C03637=1085.403,192.543,-73.156,175.423,21.883,153.539
C03638=1085.409,192.792,-73.179,175.426,21.885,153.539
C03639=1085.415,193.041,-73.202,175.428,21.886,153.539
C03640=1085.420,193.290,-73.225,175.431,21.888,153.539
C03641=1085.425,193.539,-73.248,175.433,21.890,153.539
C03642=1085.431,193.787,-73.272,175.436,21.892,153.539
C03643=1085.437,194.036,-73.295,175.438,21.893,153.539
C03644=1085.443,194.285,-73.318,175.441,21.895,153.539
C03645=1085.448,194.534,-73.342,175.443,21.897,153.539
C03646=1085.453,194.783,-73.364,175.446,21.899,153.539
C03647=1085.459,195.032,-73.387,175.448,21.900,153.539
C03648=1085.465,195.280,-73.411,175.451,21.902,153.539
C03649=1085.470,195.530,-73.435,175.453,21.904,153.539
C03650=1085.476,195.779,-73.458,175.457,21.906,153.539
C03651=1085.482,196.027,-73.481,175.459,21.907,153.539
C03652=1085.487,196.277,-73.504,175.461,21.909,153.539
C03653=1085.493,196.525,-73.528,175.464,21.911,153.539
C03654=1085.498,196.774,-73.551,175.467,21.912,153.539
C03655=1085.504,197.023,-73.574,175.469,21.914,153.539
C03656=1085.510,197.271,-73.598,175.471,21.916,153.539
C03657=1085.515,197.520,-73.621,175.474,21.917,153.539
C03658=1085.521,197.769,-73.644,175.476,21.919,153.539
C03659=1085.526,198.018,-73.667,175.479,21.921,153.539
C03660=1085.532,198.267,-73.691,175.482,21.923,153.539
C03661=1085.538,198.515,-73.714,175.485,21.925,153.539
C03662=1085.543,198.765,-73.737,175.487,21.927,153.539
C03663=1085.549,199.013,-73.761,175.490,21.928,153.539
C03664=1085.554,199.262,-73.784,175.492,21.930,153.539
C03665=1085.560,199.510,-73.808,175.495,21.932,153.539
C03666=1085.566,199.759,-73.831,175.497,21.933,153.539
C03667=1085.572,200.009,-73.855,175.500,21.935,153.539
C03668=1085.577,200.258,-73.879,175.502,21.937,153.539
C03669=1085.583,200.506,-73.902,175.505,21.938,153.539
C03670=1085.589,200.755,-73.925,175.508,21.940,153.539
C03671=1085.594,201.004,-73.949,175.511,21.942,153.538
C03672=1085.600,201.252,-73.973,175.513,21.944,153.539
C03673=1085.605,201.501,-73.996,175.516,21.945,153.539
C03674=1085.612,201.750,-74.020,175.518,21.947,153.538
C03675=1085.617,201.999,-74.043,175.521,21.949,153.538
C03676=1085.623,202.248,-74.067,175.523,21.950,153.538
C03677=1085.628,202.497,-74.090,175.526,21.952,153.538
C03678=1085.634,202.745,-74.115,175.529,21.954,153.538
C03679=1085.639,202.994,-74.138,175.532,21.956,153.538
C03680=1085.645,203.243,-74.162,175.534,21.957,153.538
C03681=1085.651,203.492,-74.185,175.537,21.959,153.538
C03682=1085.656,203.741,-74.209,175.539,21.961,153.538
C03683=1085.661,203.990,-74.233,175.542,21.963,153.538
C03684=1085.667,204.239,-74.257,175.544,21.964,153.538
C03685=1085.673,204.487,-74.281,175.548,21.966,153.538
C03686=1085.678,204.736,-74.304,175.550,21.968,153.538
C03687=1085.684,204.985,-74.328,175.553,21.970,153.538
C03688=1085.689,205.233,-74.352,175.555,21.972,153.538
C03689=1085.695,205.483,-74.376,175.558,21.973,153.538
C03690=1085.701,205.731,-74.400,175.560,21.975,153.538
C03691=1085.706,205.980,-74.424,175.564,21.977,153.538
C03692=1085.712,206.229,-74.447,175.566,21.979,153.538
C03693=1085.717,206.477,-74.471,175.568,21.981,153.538
C03694=1085.724,206.726,-74.495,175.571,21.983,153.538
C03695=1085.729,206.976,-74.519,175.574,21.984,153.538
C03696=1085.734,207.224,-74.543,175.576,21.986,153.538
C03697=1085.757,208.251,-74.642,175.658,22.028,153.535
C03698=1085.767,208.639,-74.680,175.662,22.033,153.535
C03699=1085.775,209.027,-74.718,175.666,22.037,153.535
C03700=1085.783,209.415,-74.756,175.670,22.041,153.536
C03701=1085.793,209.803,-74.795,175.673,22.045,153.536
C03702=1085.798,210.051,-74.819,175.676,22.048,153.536
C03703=1085.804,210.301,-74.843,175.678,22.050,153.536
C03704=1085.810,210.549,-74.868,175.681,22.053,153.536
C03705=1085.815,210.798,-74.892,175.684,22.056,153.537
C03706=1085.821,211.047,-74.917,175.686,22.058,153.537
C03707=1085.826,211.295,-74.942,175.689,22.061,153.537
C03708=1085.832,211.544,-74.966,175.691,22.064,153.537
C03709=1085.838,211.793,-74.990,175.694,22.067,153.538
C03710=1085.843,212.042,-75.015,175.696,22.069,153.538
C03711=1085.849,212.290,-75.040,175.699,22.072,153.538
C03712=1085.854,212.539,-75.064,175.701,22.075,153.538
C03713=1085.860,212.788,-75.089,175.704,22.077,153.538
C03714=1085.866,213.036,-75.114,175.707,22.080,153.538
C03715=1085.872,213.285,-75.138,175.709,22.083,153.539
C03716=1085.877,213.534,-75.163,175.712,22.086,153.539
C03717=1085.882,213.784,-75.188,175.714,22.088,153.539
C03718=1085.888,214.032,-75.213,175.716,22.091,153.539
C03719=1085.894,214.281,-75.238,175.720,22.094,153.539
C03720=1085.899,214.529,-75.263,175.722,22.096,153.540
C03721=1085.905,214.777,-75.287,175.725,22.099,153.540
C03722=1085.910,215.027,-75.311,175.727,22.102,153.540
C03723=1085.916,215.275,-75.336,175.730,22.105,153.540
C03724=1085.921,215.524,-75.362,175.732,22.107,153.540
C03725=1085.927,215.772,-75.387,175.734,22.110,153.541
C03726=1085.933,216.022,-75.411,175.737,22.113,153.541
C03727=1085.938,216.270,-75.436,175.740,22.115,153.541
C03728=1085.944,216.519,-75.461,175.743,22.118,153.541
C03729=1085.949,216.767,-75.486,175.745,22.121,153.541
C03730=1085.955,217.016,-75.511,175.748,22.124,153.542
C03731=1085.961,217.264,-75.536,175.750,22.126,153.542
C03732=1085.967,217.514,-75.561,175.753,22.129,153.542
C03733=1085.973,217.762,-75.586,175.755,22.132,153.542
C03734=1085.977,218.011,-75.611,175.757,22.134,153.542
C03735=1085.984,218.260,-75.636,175.761,22.137,153.543
C03736=1085.989,218.508,-75.660,175.763,22.139,153.543
C03737=1085.995,218.757,-75.686,175.766,22.143,153.543
C03738=1086.000,219.006,-75.710,175.768,22.145,153.543
C03739=1086.006,219.255,-75.736,175.771,22.148,153.543
C03740=1086.012,219.503,-75.761,175.773,22.151,153.544
C03741=1086.017,219.752,-75.785,175.776,22.153,153.544
C03742=1086.023,220.001,-75.811,175.779,22.156,153.544
C03743=1086.028,220.249,-75.836,175.782,22.159,153.544
C03744=1086.034,220.498,-75.861,175.784,22.161,153.544
C03745=1086.040,220.747,-75.886,175.786,22.164,153.544
C03746=1086.046,220.995,-75.911,175.789,22.167,153.545
C03747=1086.051,221.244,-75.937,175.791,22.169,153.545
C03748=1086.057,221.493,-75.962,175.794,22.172,153.545
C03749=1086.063,221.741,-75.987,175.797,22.175,153.545
C03750=1086.072,222.133,-76.027,175.801,22.179,153.546
C03751=1086.081,222.526,-76.066,175.805,22.183,153.546
C03752=1086.090,222.917,-76.107,175.809,22.188,153.546
C03753=1086.098,223.309,-76.146,175.813,22.192,153.547
C03754=1086.103,223.558,-76.172,175.816,22.195,153.547
C03755=1086.109,223.806,-76.197,175.818,22.197,153.547
C03756=1086.115,224.054,-76.222,175.821,22.201,153.547
C03757=1086.121,224.303,-76.248,175.824,22.203,153.547
C03758=1086.126,224.553,-76.273,175.827,22.206,153.548
C03759=1086.131,224.801,-76.298,175.829,22.209,153.548
C03760=1086.138,225.050,-76.324,175.832,22.211,153.548
C03761=1086.143,225.298,-76.350,175.834,22.214,153.548
C03762=1086.149,225.546,-76.375,175.837,22.217,153.548
C03763=1086.154,225.795,-76.401,175.839,22.219,153.548
C03764=1086.160,226.044,-76.426,175.842,22.223,153.549
C03765=1086.165,226.292,-76.452,175.845,22.225,153.549
C03766=1086.171,226.541,-76.477,175.848,22.228,153.549
C03767=1086.177,226.790,-76.503,175.850,22.231,153.549
C03768=1086.182,227.039,-76.529,175.853,22.233,153.549
C03769=1086.188,227.287,-76.554,175.855,22.236,153.550
C03770=1086.193,227.536,-76.580,175.858,22.239,153.550
C03771=1086.200,227.785,-76.605,175.860,22.241,153.550
C03772=1086.205,228.034,-76.631,175.863,22.245,153.550
C03773=1086.211,228.282,-76.656,175.866,22.247,153.551
C03774=1086.216,228.531,-76.682,175.869,22.250,153.551
C03775=1086.222,228.779,-76.707,175.871,22.252,153.551
C03776=1086.228,229.028,-76.733,175.874,22.255,153.551
C03777=1086.234,229.277,-76.760,175.876,22.258,153.551
C03778=1086.239,229.525,-76.785,175.879,22.261,153.552
C03779=1086.245,229.774,-76.811,175.881,22.263,153.552
C03780=1086.251,230.022,-76.836,175.885,22.266,153.552
C03781=1086.256,230.271,-76.862,175.887,22.269,153.552
C03782=1086.262,230.520,-76.888,175.890,22.272,153.552
C03783=1086.267,230.768,-76.913,175.892,22.274,153.552
C03784=1086.273,231.016,-76.939,175.895,22.277,153.553
C03785=1086.279,231.265,-76.965,175.898,22.280,153.553
C03786=1086.284,231.514,-76.991,175.900,22.283,153.553
C03787=1086.290,231.763,-77.017,175.903,22.285,153.553
C03788=1086.295,232.011,-77.043,175.905,22.288,153.554
C03789=1086.301,232.260,-77.069,175.909,22.291,153.554
C03790=1086.306,232.509,-77.095,175.911,22.293,153.554
C03791=1086.313,232.757,-77.120,175.914,22.297,153.554
C03792=1086.318,233.006,-77.147,175.916,22.299,153.554
C03793=1086.324,233.255,-77.173,175.919,22.302,153.555
C03794=1086.329,233.503,-77.198,175.921,22.305,153.555
C03795=1086.335,233.751,-77.224,175.924,22.307,153.555
C03796=1086.341,234.000,-77.250,175.927,22.310,153.555
C03797=1086.346,234.248,-77.277,175.930,22.313,153.555
C03798=1086.352,234.497,-77.303,175.933,22.316,153.556
C03799=1086.357,234.746,-77.329,175.935,22.319,153.556
C03800=1086.363,234.995,-77.355,175.938,22.322,153.556
C03801=1086.368,235.243,-77.381,175.940,22.324,153.556
C03802=1086.377,235.626,-77.421,175.945,22.329,153.556
C03803=1086.386,236.010,-77.462,175.948,22.333,153.557
C03804=1086.394,236.393,-77.502,175.953,22.337,153.557
C03805=1086.404,236.777,-77.542,175.957,22.341,153.557
C03806=1086.409,237.025,-77.569,175.960,22.344,153.558
C03807=1086.414,237.273,-77.595,175.962,22.347,153.558
C03808=1086.420,237.522,-77.621,175.965,22.350,153.558
C03809=1086.425,237.771,-77.647,175.968,22.353,153.558
C03810=1086.431,238.019,-77.674,175.970,22.355,153.558
C03811=1086.437,238.267,-77.700,175.973,22.359,153.559
C03812=1086.442,238.516,-77.726,175.976,22.361,153.559
C03813=1086.448,238.765,-77.753,175.979,22.364,153.559
C03814=1086.454,239.014,-77.779,175.981,22.366,153.559
C03815=1086.459,239.262,-77.806,175.984,22.369,153.559
C03816=1086.465,239.510,-77.832,175.987,22.372,153.560
C03817=1086.471,239.759,-77.858,175.989,22.375,153.560
C03818=1086.476,240.008,-77.885,175.992,22.378,153.560
C03819=1086.482,240.256,-77.912,175.994,22.380,153.560
C03820=1086.488,240.505,-77.937,175.998,22.383,153.560
C03821=1086.493,240.753,-77.964,176.001,22.386,153.561
C03822=1086.499,241.002,-77.991,176.003,22.389,153.561
C03823=1086.505,241.250,-78.017,176.006,22.391,153.561
C03824=1086.510,241.499,-78.043,176.008,22.394,153.561
C03825=1086.516,241.747,-78.070,176.011,22.397,153.561
C03826=1086.522,241.996,-78.097,176.014,22.400,153.562
C03827=1086.528,242.244,-78.123,176.016,22.403,153.562
C03828=1086.533,242.493,-78.149,176.019,22.406,153.562
C03829=1086.539,242.742,-78.176,176.022,22.408,153.562
C03830=1086.545,242.990,-78.202,176.025,22.411,153.563
C03831=1086.551,243.238,-78.229,176.028,22.414,153.563
C03832=1086.556,243.488,-78.257,176.030,22.417,153.563
C03833=1086.562,243.736,-78.283,176.033,22.420,153.563
C03834=1086.568,243.984,-78.310,176.035,22.422,153.563
C03835=1086.573,244.233,-78.336,176.038,22.425,153.564
C03836=1086.579,244.482,-78.363,176.041,22.428,153.564
C03837=1086.584,244.730,-78.390,176.043,22.431,153.564
C03838=1086.590,244.979,-78.417,176.047,22.434,153.564
C03839=1086.596,245.227,-78.443,176.050,22.437,153.565
C03840=1086.601,245.475,-78.470,176.052,22.439,153.565
C03841=1086.606,245.724,-78.497,176.055,22.443,153.565
C03842=1086.612,245.972,-78.524,176.057,22.445,153.565
C03843=1086.618,246.221,-78.550,176.060,22.448,153.565
C03844=1086.623,246.470,-78.578,176.063,22.451,153.566
C03845=1086.629,246.718,-78.604,176.065,22.454,153.566
C03846=1086.635,246.967,-78.631,176.069,22.456,153.566
C03847=1086.641,247.215,-78.658,176.071,22.460,153.566
C03848=1086.646,247.464,-78.685,176.074,22.462,153.566
C03849=1086.652,247.712,-78.712,176.077,22.465,153.567
C03850=1086.657,247.961,-78.739,176.080,22.468,153.567
C03851=1086.663,248.209,-78.766,176.082,22.471,153.567
C03852=1086.668,248.457,-78.794,176.085,22.474,153.567
C03853=1086.674,248.706,-78.820,176.087,22.476,153.568
C03854=1086.682,249.083,-78.861,176.092,22.481,153.568
C03855=1086.690,249.459,-78.902,176.096,22.486,153.568
C03856=1086.699,249.835,-78.943,176.100,22.490,153.569
C03857=1086.707,250.211,-78.984,176.105,22.494,153.569
C03858=1086.712,250.460,-79.012,176.107,22.497,153.569
C03859=1086.719,250.709,-79.039,176.110,22.500,153.569
C03860=1086.724,250.957,-79.067,176.113,22.503,153.570
C03861=1086.730,251.206,-79.093,176.115,22.506,153.570
C03862=1086.735,251.454,-79.120,176.118,22.509,153.570
C03863=1086.741,251.703,-79.147,176.121,22.512,153.570
C03864=1086.746,251.951,-79.175,176.123,22.514,153.571
C03865=1086.752,252.200,-79.202,176.126,22.518,153.571
C03866=1086.758,252.448,-79.229,176.129,22.520,153.571
C03867=1086.764,252.696,-79.257,176.132,22.523,153.571
C03868=1086.769,252.945,-79.284,176.135,22.526,153.571
C03869=1086.774,253.193,-79.311,176.138,22.529,153.572
C03870=1086.780,253.442,-79.339,176.140,22.532,153.572
C03871=1086.785,253.691,-79.366,176.143,22.535,153.572
C03872=1086.791,253.938,-79.393,176.146,22.538,153.572
C03873=1086.796,254.187,-79.421,176.148,22.540,153.573
C03874=1086.803,254.435,-79.448,176.151,22.543,153.573
C03875=1086.808,254.684,-79.476,176.154,22.546,153.573
C03876=1086.814,254.932,-79.504,176.156,22.549,153.573
C03877=1086.820,255.181,-79.531,176.160,22.552,153.574
C03878=1086.825,255.430,-79.558,176.163,22.555,153.574
C03879=1086.831,255.678,-79.585,176.165,22.558,153.574
C03880=1086.836,255.926,-79.613,176.168,22.561,153.574
C03881=1086.842,256.175,-79.641,176.171,22.564,153.575
C03882=1086.848,256.423,-79.668,176.174,22.567,153.575
C03883=1086.853,256.671,-79.695,176.176,22.569,153.575
C03884=1086.860,256.920,-79.723,176.179,22.572,153.575
C03885=1086.865,257.169,-79.750,176.182,22.575,153.575
C03886=1086.870,257.417,-79.778,176.184,22.578,153.576
C03887=1086.877,257.665,-79.806,176.187,22.581,153.576
C03888=1086.882,257.914,-79.833,176.190,22.584,153.576
C03889=1086.887,258.162,-79.861,176.193,22.586,153.576
C03890=1086.894,258.410,-79.889,176.196,22.590,153.577
C03891=1086.899,258.659,-79.916,176.199,22.592,153.577
C03892=1086.905,258.908,-79.945,176.202,22.596,153.577
C03893=1086.911,259.155,-79.972,176.204,22.598,153.577
C03894=1086.916,259.404,-79.999,176.207,22.601,153.577
C03895=1086.922,259.653,-80.028,176.210,22.604,153.578
C03896=1086.928,259.900,-80.055,176.212,22.607,153.578
C03897=1086.934,260.149,-80.083,176.216,22.609,153.578
C03898=1086.939,260.398,-80.110,176.219,22.613,153.578
C03899=1086.945,260.646,-80.138,176.222,22.616,153.579
C03900=1086.951,260.894,-80.166,176.224,22.618,153.579
C03901=1086.956,261.142,-80.194,176.227,22.621,153.579
C03902=1086.963,261.391,-80.222,176.230,22.624,153.579
C03903=1086.968,261.640,-80.249,176.233,22.627,153.579
C03904=1086.974,261.888,-80.277,176.235,22.630,153.580
C03905=1086.979,262.136,-80.305,176.238,22.633,153.580
C03906=1086.989,262.510,-80.347,176.243,22.638,153.580
C03907=1086.997,262.883,-80.390,176.247,22.641,153.581
C03908=1087.006,263.257,-80.431,176.251,22.646,153.581
C03909=1087.014,263.630,-80.474,176.256,22.650,153.581
C03910=1087.021,263.879,-80.501,176.258,22.653,153.581
C03911=1087.026,264.127,-80.529,176.261,22.656,153.582
C03912=1087.032,264.376,-80.557,176.264,22.659,153.582
C03913=1087.037,264.624,-80.585,176.266,22.662,153.582
C03914=1087.043,264.873,-80.613,176.269,22.665,153.582
C03915=1087.049,265.120,-80.642,176.272,22.668,153.583
C03916=1087.055,265.369,-80.670,176.276,22.671,153.583
C03917=1087.060,265.617,-80.698,176.279,22.674,153.583
C03918=1087.066,265.866,-80.727,176.281,22.677,153.583
C03919=1087.072,266.114,-80.755,176.284,22.680,153.584
C03920=1087.078,266.363,-80.783,176.287,22.683,153.584
C03921=1087.083,266.611,-80.811,176.290,22.686,153.584
C03922=1087.089,266.859,-80.839,176.292,22.689,153.584
C03923=1087.094,267.107,-80.867,176.295,22.691,153.585
C03924=1087.100,267.356,-80.896,176.298,22.695,153.585
C03925=1087.106,267.604,-80.924,176.301,22.698,153.585
C03926=1087.112,267.852,-80.953,176.303,22.700,153.585
C03927=1087.117,268.100,-80.981,176.306,22.703,153.586
C03928=1087.123,268.349,-81.009,176.309,22.707,153.586
C03929=1087.129,268.598,-81.037,176.312,22.710,153.586
C03930=1087.135,268.845,-81.066,176.315,22.713,153.586
C03931=1087.141,269.094,-81.094,176.318,22.715,153.587
C03932=1087.145,269.343,-81.123,176.321,22.719,153.587
C03933=1087.151,269.591,-81.152,176.324,22.721,153.587
C03934=1087.157,269.839,-81.180,176.327,22.725,153.587
C03935=1087.163,270.087,-81.208,176.329,22.727,153.588
C03936=1087.169,270.336,-81.236,176.332,22.731,153.588
C03937=1087.174,270.584,-81.265,176.335,22.733,153.588
C03938=1087.180,270.832,-81.293,176.338,22.737,153.588
C03939=1087.185,271.080,-81.323,176.341,22.740,153.589
C03940=1087.191,271.329,-81.351,176.343,22.743,153.589
C03941=1087.197,271.578,-81.379,176.346,22.745,153.589
C03942=1087.203,271.825,-81.408,176.349,22.749,153.589
C03943=1087.209,272.074,-81.436,176.352,22.752,153.590
C03944=1087.214,272.322,-81.466,176.355,22.755,153.590
C03945=1087.219,272.570,-81.494,176.357,22.758,153.590
C03946=1087.226,272.818,-81.523,176.361,22.760,153.590
C03947=1087.231,273.066,-81.551,176.364,22.764,153.591
C03948=1087.237,273.315,-81.581,176.367,22.767,153.591
C03949=1087.242,273.564,-81.609,176.370,22.770,153.591
C03950=1087.248,273.811,-81.638,176.372,22.772,153.591
C03951=1087.254,274.060,-81.666,176.375,22.776,153.592
C03952=1087.260,274.308,-81.696,176.378,22.779,153.592
C03953=1087.265,274.556,-81.723,176.381,22.782,153.592
C03954=1087.270,274.805,-81.753,176.384,22.785,153.593
C03955=1087.276,275.054,-81.781,176.387,22.789,153.593
C03956=1087.282,275.301,-81.810,176.389,22.791,153.593
C03957=1087.288,275.549,-81.840,176.392,22.794,153.593
C03958=1087.296,275.926,-81.883,176.397,22.799,153.594
C03959=1087.304,276.302,-81.927,176.401,22.804,153.594
C03960=1087.313,276.678,-81.970,176.406,22.808,153.594
C03961=1087.322,277.055,-82.015,176.409,22.813,153.595
C03962=1087.328,277.303,-82.044,176.412,22.816,153.595
C03963=1087.333,277.552,-82.073,176.415,22.819,153.596
C03964=1087.339,277.800,-82.102,176.419,22.822,153.596
C03965=1087.345,278.049,-82.131,176.422,22.825,153.596
C03966=1087.351,278.296,-82.160,176.425,22.828,153.596
C03967=1087.356,278.544,-82.190,176.427,22.831,153.597
C03968=1087.362,278.793,-82.218,176.430,22.834,153.597
C03969=1087.368,279.042,-82.247,176.433,22.838,153.597
C03970=1087.373,279.289,-82.276,176.436,22.841,153.597
C03971=1087.379,279.537,-82.306,176.439,22.844,153.598
C03972=1087.385,279.786,-82.335,176.442,22.847,153.598
C03973=1087.390,280.034,-82.364,176.445,22.851,153.598
C03974=1087.396,280.281,-82.393,176.447,22.853,153.598
C03975=1087.402,280.530,-82.423,176.450,22.856,153.599
C03976=1087.408,280.779,-82.451,176.453,22.859,153.599
C03977=1087.413,281.027,-82.481,176.456,22.862,153.599
C03978=1087.419,281.275,-82.510,176.459,22.866,153.600
C03979=1087.424,281.523,-82.539,176.462,22.869,153.600
C03980=1087.431,281.771,-82.568,176.465,22.872,153.600
C03981=1087.436,282.020,-82.598,176.467,22.875,153.601
C03982=1087.442,282.268,-82.627,176.470,22.878,153.601
C03983=1087.448,282.516,-82.656,176.473,22.881,153.601
C03984=1087.453,282.764,-82.686,176.476,22.884,153.601
C03985=1087.458,283.012,-82.715,176.479,22.888,153.602
C03986=1087.464,283.260,-82.746,176.482,22.891,153.602
C03987=1087.470,283.508,-82.775,176.485,22.894,153.602
C03988=1087.476,283.757,-82.804,176.488,22.897,153.603
C03989=1087.481,284.005,-82.834,176.491,22.900,153.603
C03990=1087.487,284.253,-82.863,176.493,22.903,153.603
C03991=1087.492,284.501,-82.892,176.496,22.907,153.604
C03992=1087.498,284.749,-82.922,176.499,22.910,153.604
C03993=1087.503,284.998,-82.952,176.502,22.913,153.604
C03994=1087.510,285.245,-82.981,176.505,22.917,153.604
C03995=1087.516,285.494,-83.011,176.508,22.920,153.605
C03996=1087.521,285.742,-83.041,176.511,22.923,153.605
C03997=1087.527,285.990,-83.070,176.514,22.926,153.605
C03998=1087.533,286.238,-83.100,176.517,22.929,153.606
C03999=1087.538,286.486,-83.129,176.519,22.932,153.606
C04000=1087.544,286.734,-83.159,176.522,22.935,153.606
C04001=1087.549,286.983,-83.188,176.525,22.939,153.606
C04002=1087.556,287.230,-83.218,176.528,22.942,153.607
C04003=1087.561,287.479,-83.248,176.531,22.945,153.607
C04004=1087.567,287.727,-83.278,176.534,22.948,153.607
C04005=1087.572,287.975,-83.308,176.537,22.951,153.608
C04006=1087.579,288.223,-83.337,176.540,22.955,153.608
C04007=1087.584,288.472,-83.367,176.544,22.958,153.608
C04008=1087.590,288.719,-83.397,176.547,22.961,153.608
C04009=1087.596,288.968,-83.427,176.549,22.965,153.609
C04010=1087.604,289.354,-83.473,176.554,22.969,153.609
C04011=1087.613,289.740,-83.520,176.558,22.974,153.610
C04012=1087.622,290.125,-83.566,176.563,22.979,153.610
C04013=1087.631,290.511,-83.613,176.567,22.984,153.611
C04014=1087.636,290.760,-83.643,176.570,22.988,153.611
C04015=1087.642,291.007,-83.673,176.573,22.991,153.611
C04016=1087.648,291.256,-83.703,176.576,22.994,153.612
C04017=1087.654,291.504,-83.733,176.579,22.998,153.612
C04018=1087.660,291.752,-83.762,176.582,23.001,153.612
C04019=1087.666,292.000,-83.792,176.585,23.004,153.613
C04020=1087.671,292.248,-83.822,176.588,23.007,153.613
C04021=1087.677,292.496,-83.852,176.591,23.011,153.613
C04022=1087.682,292.744,-83.883,176.594,23.014,153.614
C04023=1087.688,292.992,-83.913,176.597,23.017,153.614
C04024=1087.694,293.241,-83.944,176.599,23.020,153.614
C04025=1087.700,293.489,-83.974,176.602,23.024,153.615
C04026=1087.705,293.737,-84.004,176.605,23.027,153.615
C04027=1087.711,293.985,-84.034,176.608,23.030,153.615
C04028=1087.717,294.233,-84.064,176.611,23.033,153.615
C04029=1087.723,294.481,-84.095,176.614,23.037,153.616
C04030=1087.728,294.729,-84.124,176.617,23.040,153.616
C04031=1087.734,294.977,-84.155,176.620,23.043,153.616
C04032=1087.740,295.225,-84.185,176.623,23.046,153.617
C04033=1087.746,295.473,-84.215,176.626,23.050,153.617
C04034=1087.751,295.721,-84.245,176.629,23.053,153.617
C04035=1087.757,295.969,-84.275,176.632,23.057,153.618
C04036=1087.763,296.218,-84.307,176.635,23.060,153.618
C04037=1087.769,296.466,-84.337,176.638,23.063,153.618
C04038=1087.774,296.713,-84.367,176.641,23.067,153.619
C04039=1087.780,296.961,-84.398,176.644,23.070,153.619
C04040=1087.786,297.209,-84.428,176.647,23.073,153.619
C04041=1087.791,297.458,-84.458,176.650,23.077,153.620
C04042=1087.797,297.706,-84.489,176.653,23.080,153.620
C04043=1087.803,297.954,-84.519,176.656,23.084,153.620
C04044=1087.809,298.202,-84.550,176.659,23.087,153.621
C04045=1087.814,298.450,-84.581,176.662,23.090,153.621
C04046=1087.820,298.698,-84.611,176.665,23.094,153.621
C04047=1087.825,298.946,-84.642,176.667,23.097,153.622
C04048=1087.831,299.194,-84.672,176.670,23.101,153.622
C04049=1087.837,299.442,-84.703,176.673,23.104,153.623
C04050=1087.842,299.690,-84.734,176.676,23.108,153.623
C04051=1087.847,299.938,-84.764,176.679,23.111,153.623
C04052=1087.853,300.186,-84.796,176.682,23.115,153.624
C04053=1087.859,300.434,-84.826,176.685,23.118,153.624
C04054=1087.864,300.682,-84.857,176.688,23.121,153.624
C04055=1087.870,300.930,-84.888,176.691,23.125,153.625
C04056=1087.876,301.177,-84.918,176.694,23.128,153.625
C04057=1087.881,301.426,-84.949,176.697,23.132,153.626
C04058=1087.887,301.674,-84.980,176.700,23.135,153.626
C04059=1087.893,301.922,-85.011,176.703,23.139,153.626
C04060=1087.899,302.169,-85.042,176.706,23.142,153.627
C04061=1087.904,302.418,-85.073,176.708,23.146,153.627
C04062=1087.913,302.818,-85.122,176.714,23.152,153.628
C04063=1087.922,303.217,-85.172,176.718,23.157,153.628
C04064=1087.932,303.618,-85.222,176.723,23.163,153.629
C04065=1087.940,304.018,-85.272,176.728,23.168,153.629
C04066=1087.946,304.265,-85.303,176.731,23.172,153.630
C04067=1087.952,304.514,-85.335,176.734,23.175,153.630
C04068=1087.958,304.762,-85.365,176.737,23.179,153.631
C04069=1087.963,305.010,-85.396,176.740,23.183,153.631
C04070=1087.969,305.257,-85.427,176.743,23.186,153.631
C04071=1087.975,305.506,-85.458,176.746,23.189,153.632
C04072=1087.981,305.753,-85.489,176.749,23.193,153.632
C04073=1087.986,306.001,-85.520,176.752,23.196,153.632
C04074=1087.992,306.250,-85.552,176.755,23.200,153.633
C04075=1087.998,306.497,-85.583,176.758,23.203,153.633
C04076=1088.003,306.745,-85.614,176.761,23.207,153.634
C04077=1088.010,306.993,-85.645,176.764,23.210,153.634
C04078=1088.015,307.241,-85.676,176.767,23.214,153.634
C04079=1088.021,307.488,-85.707,176.769,23.217,153.635
C04080=1088.026,307.737,-85.738,176.773,23.221,153.635
C04081=1088.032,307.985,-85.770,176.776,23.224,153.635
C04082=1088.039,308.233,-85.802,176.779,23.228,153.636
C04083=1088.044,308.481,-85.832,176.782,23.232,153.636
C04084=1088.050,308.728,-85.864,176.785,23.235,153.637
C04085=1088.055,308.977,-85.895,176.788,23.239,153.637
C04086=1088.061,309.224,-85.927,176.791,23.242,153.637
C04087=1088.068,309.472,-85.958,176.794,23.246,153.638
C04088=1088.073,309.720,-85.989,176.797,23.249,153.638
C04089=1088.078,309.968,-86.021,176.800,23.253,153.639
C04090=1088.085,310.216,-86.052,176.802,23.256,153.639
C04091=1088.090,310.464,-86.083,176.806,23.260,153.639
C04092=1088.096,310.712,-86.115,176.809,23.264,153.640
C04093=1088.102,310.959,-86.146,176.812,23.267,153.640
C04094=1088.108,311.208,-86.177,176.815,23.271,153.641
C04095=1088.113,311.456,-86.209,176.818,23.274,153.641
C04096=1088.120,311.704,-86.240,176.821,23.278,153.641
C04097=1088.125,311.951,-86.272,176.824,23.281,153.642
C04098=1088.131,312.199,-86.304,176.827,23.285,153.642
C04099=1088.136,312.447,-86.335,176.830,23.288,153.642
C04100=1088.143,312.695,-86.366,176.833,23.292,153.643
C04101=1088.149,312.944,-86.399,176.836,23.296,153.643
C04102=1088.154,313.191,-86.430,176.839,23.300,153.644
C04103=1088.161,313.439,-86.462,176.842,23.303,153.644
C04104=1088.166,313.686,-86.493,176.845,23.306,153.644
C04105=1088.172,313.935,-86.525,176.848,23.310,153.645
C04106=1088.177,314.183,-86.556,176.851,23.314,153.645
C04107=1088.184,314.431,-86.588,176.854,23.317,153.646
C04108=1088.190,314.679,-86.620,176.857,23.321,153.646
C04109=1088.196,314.926,-86.651,176.861,23.325,153.646
C04110=1088.201,315.175,-86.683,176.863,23.328,153.647
C04111=1088.207,315.422,-86.715,176.866,23.332,153.647
C04112=1088.213,315.670,-86.747,176.869,23.336,153.648
C04113=1088.218,315.918,-86.779,176.872,23.340,153.648
C04114=1088.225,316.226,-86.819,176.875,23.344,153.649
C04115=1088.232,316.532,-86.859,176.879,23.349,153.649
C04116=1088.239,316.841,-86.898,176.884,23.354,153.650
C04117=1088.246,317.147,-86.938,176.887,23.359,153.651
C04118=1088.252,317.395,-86.970,176.890,23.362,153.651
C04119=1088.258,317.643,-87.001,176.893,23.366,153.651
C04120=1088.263,317.891,-87.034,176.896,23.370,153.652
C04121=1088.269,318.138,-87.066,176.899,23.373,153.652
C04122=1088.275,318.387,-87.098,176.901,23.377,153.653
C04123=1088.281,318.635,-87.130,176.905,23.381,153.653
C04124=1088.286,318.882,-87.162,176.908,23.385,153.654
C04125=1088.292,319.130,-87.194,176.911,23.389,153.654
C04126=1088.297,319.378,-87.227,176.914,23.392,153.654
C04127=1088.303,319.626,-87.259,176.916,23.396,153.655
C04128=1088.309,319.874,-87.291,176.919,23.400,153.655
C04129=1088.314,320.122,-87.323,176.923,23.404,153.656
C04130=1088.321,320.369,-87.356,176.926,23.408,153.656
C04131=1088.326,320.618,-87.388,176.929,23.412,153.657
C04132=1088.331,320.865,-87.420,176.932,23.415,153.657
C04133=1088.337,321.113,-87.453,176.934,23.419,153.658
C04134=1088.343,321.361,-87.485,176.938,23.424,153.658
C04135=1088.348,321.609,-87.517,176.941,23.427,153.659
C04136=1088.354,321.856,-87.550,176.944,23.431,153.659
C04137=1088.360,322.105,-87.582,176.947,23.435,153.660
C04138=1088.366,322.352,-87.614,176.949,23.439,153.660
C04139=1088.371,322.600,-87.647,176.953,23.443,153.661
C04140=1088.378,322.848,-87.679,176.956,23.447,153.661
C04141=1088.384,323.096,-87.711,176.959,23.450,153.662
C04142=1088.391,323.439,-87.756,176.963,23.456,153.662
C04143=1088.399,323.783,-87.801,176.967,23.461,153.663
C04144=1088.408,324.126,-87.847,176.971,23.466,153.664
C04145=1088.415,324.469,-87.891,176.975,23.472,153.664
C04146=1088.421,324.717,-87.925,176.979,23.476,153.665
C04147=1088.427,324.965,-87.957,176.982,23.480,153.665
C04148=1088.433,325.212,-87.989,176.985,23.484,153.666
C04149=1088.438,325.460,-88.022,176.987,23.488,153.666
C04150=1088.444,325.708,-88.054,176.990,23.491,153.667
C04151=1088.450,325.955,-88.087,176.994,23.496,153.667
C04152=1088.456,326.204,-88.120,176.997,23.499,153.668
C04153=1088.462,326.452,-88.152,177.000,23.504,153.668
C04154=1088.468,326.699,-88.185,177.002,23.507,153.669
C04155=1088.473,326.948,-88.218,177.006,23.512,153.669
C04156=1088.479,327.195,-88.250,177.009,23.515,153.670
C04157=1088.485,327.442,-88.283,177.012,23.519,153.670
C04158=1088.491,327.690,-88.316,177.015,23.523,153.671
C04159=1088.497,327.938,-88.348,177.018,23.528,153.671
C04160=1088.502,328.186,-88.382,177.021,23.531,153.672
C04161=1088.509,328.434,-88.414,177.024,23.535,153.672
C04162=1088.515,328.681,-88.447,177.027,23.539,153.673
C04163=1088.521,328.929,-88.480,177.030,23.543,153.673
C04164=1088.527,329.177,-88.513,177.033,23.547,153.673
C04165=1088.532,329.425,-88.546,177.036,23.551,153.674
C04166=1088.542,329.821,-88.598,177.041,23.557,153.675
C04167=1088.551,330.217,-88.650,177.046,23.564,153.676
C04168=1088.561,330.613,-88.704,177.051,23.571,153.676
C04169=1088.570,331.009,-88.757,177.056,23.577,153.677
C04170=1088.577,331.256,-88.789,177.059,23.581,153.678
C04171=1088.582,331.504,-88.823,177.062,23.585,153.678
C04172=1088.588,331.752,-88.855,177.065,23.589,153.679
C04173=1088.594,332.000,-88.889,177.068,23.593,153.679
C04174=1088.600,332.248,-88.922,177.071,23.597,153.680
C04175=1088.606,332.495,-88.955,177.074,23.601,153.680
C04176=1088.611,332.743,-88.988,177.077,23.605,153.681
C04177=1088.617,332.991,-89.021,177.080,23.609,153.681
C04178=1088.623,333.239,-89.055,177.083,23.614,153.682
C04179=1088.629,333.486,-89.088,177.087,23.618,153.683
C04180=1088.635,333.734,-89.122,177.089,23.622,153.683
C04181=1088.640,333.982,-89.155,177.092,23.626,153.684
C04182=1088.646,334.230,-89.188,177.096,23.631,153.684
C04183=1088.652,334.477,-89.221,177.098,23.635,153.685
C04184=1088.658,334.725,-89.254,177.101,23.639,153.685
C04185=1088.664,334.972,-89.288,177.105,23.643,153.686
C04186=1088.669,335.220,-89.322,177.108,23.647,153.687
C04187=1088.675,335.468,-89.355,177.110,23.652,153.687
C04188=1088.681,335.716,-89.388,177.114,23.656,153.688
C04189=1088.687,335.963,-89.422,177.117,23.660,153.688
C04190=1088.692,336.211,-89.455,177.119,23.664,153.689
C04191=1088.698,336.459,-89.489,177.123,23.669,153.689
C04192=1088.704,336.706,-89.523,177.126,23.673,153.690
C04193=1088.711,336.954,-89.556,177.129,23.677,153.690
C04194=1088.716,337.202,-89.589,177.132,23.681,153.691
C04195=1088.722,337.450,-89.623,177.135,23.685,153.692
C04196=1088.728,337.697,-89.656,177.139,23.690,153.692
C04197=1088.733,337.945,-89.690,177.141,23.694,153.693
C04198=1088.739,338.193,-89.724,177.144,23.699,153.693
C04199=1088.745,338.441,-89.757,177.148,23.703,153.694
C04200=1088.750,338.688,-89.791,177.150,23.707,153.694
C04201=1088.757,338.936,-89.825,177.153,23.711,153.695
C04202=1088.762,339.184,-89.859,177.157,23.716,153.696
C04203=1088.768,339.432,-89.892,177.159,23.720,153.696
C04204=1088.774,339.679,-89.926,177.163,23.725,153.697
C04205=1088.780,339.926,-89.960,177.166,23.729,153.697
C04206=1088.785,340.174,-89.994,177.168,23.733,153.698
C04207=1088.791,340.421,-90.028,177.172,23.738,153.699
C04208=1088.797,340.669,-90.061,177.175,23.742,153.699
C04209=1088.803,340.917,-90.096,177.178,23.747,153.700
C04210=1088.809,341.165,-90.130,177.181,23.751,153.700
C04211=1088.815,341.412,-90.163,177.184,23.755,153.701
C04212=1088.820,341.660,-90.197,177.187,23.760,153.702
C04213=1088.826,341.907,-90.231,177.190,23.764,153.702
C04214=1088.832,342.156,-90.265,177.194,23.769,153.703
C04215=1088.838,342.403,-90.299,177.196,23.773,153.704
C04216=1088.844,342.650,-90.333,177.200,23.778,153.704
C04217=1088.850,342.897,-90.367,177.203,23.782,153.705
C04218=1088.859,343.288,-90.421,177.207,23.789,153.706
C04219=1088.868,343.679,-90.474,177.212,23.797,153.707
C04220=1088.878,344.068,-90.528,177.217,23.803,153.708
C04221=1088.887,344.459,-90.581,177.222,23.811,153.709
C04222=1088.892,344.706,-90.616,177.225,23.815,153.710
C04223=1088.899,344.954,-90.650,177.228,23.820,153.710
C04224=1088.905,345.202,-90.684,177.231,23.824,153.711
C04225=1088.910,345.449,-90.718,177.234,23.829,153.711
C04226=1088.916,345.696,-90.752,177.237,23.833,153.712
C04227=1088.922,345.944,-90.787,177.241,23.838,153.713
C04228=1088.928,346.192,-90.821,177.243,23.843,153.713
C04229=1088.934,346.439,-90.855,177.247,23.847,153.714
C04230=1088.939,346.687,-90.891,177.250,23.852,153.715
C04231=1088.945,346.935,-90.925,177.253,23.856,153.715
C04232=1088.951,347.182,-90.959,177.256,23.861,153.716
C04233=1088.957,347.430,-90.994,177.259,23.866,153.717
C04234=1088.963,347.677,-91.028,177.262,23.870,153.717
C04235=1088.969,347.925,-91.062,177.265,23.875,153.718
C04236=1088.975,348.172,-91.097,177.268,23.879,153.719
C04237=1088.981,348.420,-91.132,177.272,23.884,153.719
C04238=1088.986,348.667,-91.166,177.274,23.889,153.720
C04239=1088.992,348.915,-91.201,177.278,23.894,153.721
C04240=1088.998,349.163,-91.235,177.280,23.898,153.721
C04241=1089.003,349.410,-91.269,177.284,23.903,153.722
C04242=1089.010,349.658,-91.304,177.286,23.908,153.723
C04243=1089.016,349.905,-91.338,177.290,23.913,153.724
C04244=1089.021,350.153,-91.373,177.293,23.917,153.724
C04245=1089.027,350.400,-91.408,177.296,23.922,153.725
C04246=1089.033,350.647,-91.443,177.299,23.927,153.726
C04247=1089.039,350.895,-91.477,177.302,23.932,153.726
C04248=1089.044,351.143,-91.512,177.305,23.936,153.727
C04249=1089.051,351.390,-91.547,177.308,23.941,153.728
C04250=1089.057,351.638,-91.581,177.311,23.946,153.728
C04251=1089.062,351.885,-91.617,177.315,23.951,153.729
C04252=1089.069,352.133,-91.651,177.317,23.956,153.730
C04253=1089.074,352.380,-91.686,177.321,23.961,153.731
C04254=1089.081,352.628,-91.721,177.324,23.965,153.731
C04255=1089.086,352.875,-91.755,177.327,23.970,153.732
C04256=1089.093,353.122,-91.791,177.330,23.975,153.733
C04257=1089.098,353.370,-91.825,177.333,23.980,153.734
C04258=1089.104,353.618,-91.861,177.336,23.985,153.734
C04259=1089.110,353.865,-91.895,177.339,23.989,153.735
C04260=1089.116,354.113,-91.931,177.342,23.995,153.736
C04261=1089.122,354.360,-91.965,177.345,23.999,153.736
C04262=1089.128,354.608,-92.000,177.348,24.004,153.737
C04263=1089.133,354.855,-92.036,177.352,24.010,153.738
C04264=1089.139,355.103,-92.070,177.354,24.014,153.739
C04265=1089.145,355.350,-92.106,177.358,24.019,153.739
C04266=1089.151,355.598,-92.141,177.360,24.024,153.740
C04267=1089.156,355.845,-92.176,177.364,24.029,153.741
C04268=1089.163,356.092,-92.211,177.367,24.034,153.742
C04269=1089.168,356.339,-92.246,177.370,24.039,153.742
C04270=1089.178,356.732,-92.302,177.374,24.047,153.744
C04271=1089.187,357.126,-92.358,177.380,24.055,153.745
C04272=1089.196,357.518,-92.414,177.385,24.063,153.746
C04273=1089.205,357.911,-92.470,177.389,24.071,153.747
C04274=1089.212,358.159,-92.505,177.393,24.076,153.748
C04275=1089.217,358.405,-92.541,177.396,24.081,153.749
C04276=1089.223,358.653,-92.576,177.399,24.086,153.750
C04277=1089.229,358.901,-92.612,177.402,24.091,153.750
C04278=1089.236,359.147,-92.647,177.406,24.097,153.751
C04279=1089.241,359.396,-92.682,177.408,24.102,153.752
C04280=1089.247,359.643,-92.718,177.411,24.107,153.753
C04281=1089.253,359.890,-92.753,177.414,24.112,153.754
C04282=1089.259,360.138,-92.789,177.417,24.117,153.754
C04283=1089.265,360.385,-92.823,177.421,24.122,153.755
C04284=1089.271,360.632,-92.859,177.423,24.127,153.756
C04285=1089.277,360.880,-92.895,177.427,24.133,153.757
C04286=1089.283,361.127,-92.930,177.430,24.138,153.758
C04287=1089.289,361.374,-92.967,177.433,24.143,153.759
C04288=1089.295,361.622,-93.002,177.436,24.148,153.759
C04289=1089.300,361.869,-93.038,177.439,24.154,153.760
C04290=1089.306,362.116,-93.074,177.442,24.159,153.761
C04291=1089.312,362.364,-93.109,177.445,24.164,153.762
C04292=1089.318,362.611,-93.145,177.449,24.169,153.763
C04293=1089.324,362.859,-93.180,177.451,24.174,153.764
C04294=1089.330,363.106,-93.217,177.455,24.180,153.764
C04295=1089.336,363.354,-93.253,177.458,24.186,153.765
C04296=1089.342,363.601,-93.288,177.460,24.191,153.766
C04297=1089.348,363.848,-93.324,177.464,24.196,153.767
C04298=1089.354,364.095,-93.360,177.467,24.201,153.768
C04299=1089.359,364.342,-93.395,177.471,24.207,153.769
C04300=1089.365,364.590,-93.431,177.473,24.212,153.770
C04301=1089.371,364.838,-93.467,177.476,24.217,153.770
C04302=1089.378,365.085,-93.503,177.480,24.223,153.771
C04303=1089.383,365.332,-93.539,177.482,24.228,153.772
C04304=1089.390,365.579,-93.575,177.486,24.234,153.773
C04305=1089.396,365.826,-93.611,177.489,24.239,153.774
C04306=1089.402,366.074,-93.647,177.492,24.245,153.775
C04307=1089.408,366.321,-93.683,177.495,24.250,153.776
C04308=1089.413,366.568,-93.719,177.498,24.256,153.777
C04309=1089.419,366.815,-93.755,177.501,24.261,153.777
C04310=1089.425,367.063,-93.791,177.504,24.266,153.778
C04311=1089.431,367.310,-93.828,177.507,24.272,153.779
C04312=1089.436,367.557,-93.864,177.510,24.278,153.780
C04313=1089.442,367.804,-93.900,177.514,24.283,153.781
C04314=1089.448,368.052,-93.936,177.516,24.289,153.782
C04315=1089.455,368.299,-93.972,177.519,24.295,153.783
C04316=1089.460,368.547,-94.009,177.523,24.300,153.784
C04317=1089.466,368.794,-94.045,177.526,24.306,153.785
C04318=1089.472,369.041,-94.081,177.528,24.311,153.786
C04319=1089.478,369.288,-94.117,177.532,24.317,153.787
C04320=1089.484,369.536,-94.154,177.535,24.322,153.787
C04321=1089.490,369.783,-94.190,177.538,24.328,153.788
C04322=1089.500,370.190,-94.250,177.544,24.337,153.790
C04323=1089.510,370.599,-94.311,177.549,24.347,153.792
C04324=1089.520,371.007,-94.371,177.553,24.356,153.793
C04325=1089.529,371.416,-94.431,177.558,24.366,153.795
C04326=1089.535,371.663,-94.467,177.561,24.371,153.796
C04327=1089.542,371.910,-94.504,177.565,24.377,153.797
C04328=1089.547,372.158,-94.541,177.568,24.383,153.798
C04329=1089.554,372.405,-94.577,177.571,24.389,153.799
C04330=1089.559,372.652,-94.614,177.574,24.394,153.800
C04331=1089.565,372.899,-94.651,177.577,24.400,153.801
C04332=1089.572,373.146,-94.687,177.580,24.406,153.801
C04333=1089.577,373.393,-94.724,177.584,24.412,153.802
C04334=1089.584,373.640,-94.760,177.587,24.418,153.804
C04335=1089.590,373.888,-94.797,177.590,24.424,153.804
C04336=1089.596,374.135,-94.834,177.592,24.429,153.805
C04337=1089.602,374.382,-94.870,177.596,24.435,153.807
C04338=1089.608,374.629,-94.907,177.599,24.441,153.807
C04339=1089.613,374.877,-94.944,177.602,24.447,153.808
C04340=1089.620,375.124,-94.981,177.605,24.453,153.810
C04341=1089.625,375.371,-95.018,177.608,24.459,153.811
C04342=1089.632,375.618,-95.054,177.611,24.465,153.812
C04343=1089.637,375.865,-95.092,177.614,24.471,153.813
C04344=1089.643,376.112,-95.129,177.617,24.477,153.814
C04345=1089.649,376.359,-95.166,177.620,24.483,153.815
C04346=1089.655,376.607,-95.203,177.624,24.489,153.816
C04347=1089.661,376.854,-95.240,177.627,24.495,153.817
C04348=1089.667,377.100,-95.277,177.630,24.501,153.818
C04349=1089.673,377.348,-95.314,177.633,24.508,153.819
C04350=1089.679,377.595,-95.350,177.636,24.514,153.820
C04351=1089.685,377.842,-95.388,177.639,24.519,153.821
C04352=1089.691,378.089,-95.425,177.642,24.526,153.822
C04353=1089.697,378.336,-95.462,177.645,24.532,153.823
C04354=1089.703,378.583,-95.499,177.648,24.538,153.824
C04355=1089.708,378.830,-95.536,177.651,24.544,153.825
C04356=1089.714,379.077,-95.574,177.655,24.551,153.826
C04357=1089.721,379.325,-95.611,177.658,24.557,153.827
C04358=1089.727,379.572,-95.648,177.661,24.563,153.829
C04359=1089.733,379.819,-95.686,177.664,24.569,153.830
C04360=1089.739,380.066,-95.722,177.667,24.576,153.831
C04361=1089.745,380.313,-95.760,177.670,24.582,153.832
C04362=1089.751,380.559,-95.798,177.674,24.588,153.833
C04363=1089.757,380.807,-95.835,177.676,24.594,153.834
C04364=1089.764,381.054,-95.872,177.679,24.600,153.835
C04365=1089.769,381.301,-95.909,177.682,24.606,153.836
C04366=1089.775,381.548,-95.947,177.685,24.613,153.837
C04367=1089.781,381.795,-95.985,177.688,24.619,153.838
C04368=1089.788,382.042,-96.021,177.692,24.625,153.840
C04369=1089.794,382.289,-96.059,177.695,24.632,153.841
C04370=1089.800,382.536,-96.097,177.698,24.638,153.842
C04371=1089.806,382.783,-96.134,177.701,24.645,153.843
C04372=1089.811,383.030,-96.172,177.704,24.651,153.844
C04373=1089.817,383.277,-96.210,177.707,24.658,153.845
C04374=1089.823,383.496,-96.243,177.711,24.664,153.846
C04375=1089.828,383.713,-96.276,177.713,24.669,153.847
C04376=1089.834,383.931,-96.310,177.715,24.675,153.848
C04377=1089.838,384.149,-96.342,177.719,24.681,153.849
C04378=1089.844,384.367,-96.376,177.721,24.687,153.850
C04379=1089.850,384.585,-96.410,177.724,24.693,153.852
C04380=1089.854,384.803,-96.442,177.727,24.698,153.852
C04381=1089.860,385.021,-96.476,177.729,24.704,153.854
C04382=1089.866,385.268,-96.514,177.732,24.711,153.855
C04383=1089.872,385.515,-96.552,177.736,24.718,153.856
C04384=1089.878,385.762,-96.590,177.739,24.724,153.857
C04385=1089.884,386.009,-96.628,177.742,24.731,153.858
C04386=1089.890,386.256,-96.665,177.745,24.737,153.860
C04387=1089.896,386.503,-96.703,177.748,24.744,153.861
C04388=1089.902,386.750,-96.741,177.751,24.751,153.862
C04389=1089.908,386.997,-96.779,177.754,24.757,153.863
C04390=1089.914,387.244,-96.817,177.757,24.764,153.864
C04391=1089.921,387.491,-96.855,177.760,24.771,153.866
C04392=1089.926,387.738,-96.893,177.763,24.778,153.867
C04393=1089.932,387.985,-96.931,177.766,24.784,153.868
C04394=1089.938,388.232,-96.969,177.770,24.791,153.869
C04395=1089.945,388.478,-97.008,177.773,24.798,153.871
C04396=1089.950,388.725,-97.045,177.776,24.804,153.872
C04397=1089.957,388.973,-97.083,177.779,24.812,153.873
C04398=1089.963,389.219,-97.121,177.783,24.819,153.874
C04399=1089.969,389.465,-97.160,177.786,24.825,153.876
C04400=1089.975,389.713,-97.198,177.789,24.832,153.877
C04401=1089.981,389.960,-97.236,177.792,24.839,153.878
C04402=1089.987,390.207,-97.274,177.795,24.846,153.879
C04403=1089.993,390.453,-97.313,177.798,24.853,153.881
C04404=1090.000,390.701,-97.351,177.801,24.860,153.882
C04405=1090.006,390.947,-97.389,177.804,24.867,153.883
C04406=1090.012,391.195,-97.428,177.807,24.874,153.885
C04407=1090.018,391.442,-97.466,177.811,24.881,153.886
C04408=1090.025,391.688,-97.505,177.814,24.888,153.887
C04409=1090.031,391.935,-97.542,177.817,24.895,153.889
C04410=1090.037,392.182,-97.582,177.820,24.902,153.890
C04411=1090.043,392.429,-97.620,177.823,24.909,153.891
C04412=1090.049,392.676,-97.658,177.826,24.916,153.893
C04413=1090.055,392.923,-97.697,177.828,24.923,153.894
C04414=1090.061,393.170,-97.736,177.832,24.931,153.895
C04415=1090.067,393.416,-97.773,177.835,24.938,153.897
C04416=1090.073,393.664,-97.813,177.838,24.945,153.898
C04417=1090.080,393.910,-97.851,177.841,24.952,153.899
C04418=1090.085,394.157,-97.890,177.844,24.959,153.901
C04419=1090.091,394.404,-97.928,177.848,24.967,153.902
C04420=1090.098,394.651,-97.968,177.851,24.974,153.903
C04421=1090.103,394.897,-98.006,177.854,24.982,153.905
C04422=1090.110,395.144,-98.044,177.857,24.989,153.906
C04423=1090.116,395.391,-98.084,177.860,24.996,153.907
C04424=1090.122,395.638,-98.122,177.863,25.003,153.909
C04425=1090.128,395.885,-98.161,177.867,25.011,153.910
C04426=1090.134,396.132,-98.200,177.869,25.018,153.912
C04427=1090.141,396.379,-98.239,177.872,25.026,153.913
C04428=1090.147,396.626,-98.278,177.875,25.033,153.915
C04429=1090.153,396.872,-98.317,177.879,25.041,153.916
C04430=1090.159,397.097,-98.353,177.881,25.047,153.917
C04431=1090.164,397.322,-98.388,177.884,25.054,153.919
C04432=1090.169,397.546,-98.423,177.887,25.061,153.920
C04433=1090.175,397.771,-98.459,177.890,25.068,153.921
C04434=1090.181,397.996,-98.494,177.893,25.075,153.923
C04435=1090.186,398.221,-98.530,177.896,25.082,153.924
C04436=1090.192,398.445,-98.566,177.899,25.089,153.925
C04437=1090.198,398.670,-98.601,177.902,25.096,153.927
C04438=1090.204,398.917,-98.641,177.904,25.103,153.928
C04439=1090.210,399.163,-98.679,177.907,25.111,153.930
C04440=1090.216,399.410,-98.719,177.911,25.119,153.931
C04441=1090.222,399.657,-98.758,177.914,25.126,153.932
C04442=1090.228,399.905,-98.798,177.917,25.134,153.934
C04443=1090.234,400.151,-98.836,177.920,25.142,153.936
C04444=1090.240,400.398,-98.876,177.923,25.150,153.937
C04445=1090.246,400.645,-98.915,177.926,25.157,153.938
C04446=1090.253,400.892,-98.955,177.929,25.165,153.940
C04447=1090.258,401.138,-98.994,177.933,25.173,153.942
C04448=1090.265,401.385,-99.033,177.935,25.181,153.943
C04449=1090.271,401.632,-99.073,177.938,25.189,153.945
C04450=1090.278,401.878,-99.113,177.942,25.197,153.946
C04451=1090.284,402.126,-99.152,177.945,25.205,153.948
C04452=1090.289,402.372,-99.191,177.949,25.213,153.949
C04453=1090.296,402.619,-99.231,177.951,25.221,153.951
C04454=1090.302,402.866,-99.271,177.954,25.229,153.952
C04455=1090.308,403.112,-99.310,177.958,25.237,153.954
C04456=1090.315,403.359,-99.350,177.961,25.245,153.956
C04457=1090.321,403.606,-99.389,177.963,25.253,153.957
C04458=1090.327,403.853,-99.429,177.967,25.261,153.959
C04459=1090.333,404.100,-99.469,177.970,25.269,153.960
C04460=1090.340,404.346,-99.509,177.974,25.278,153.962
C04461=1090.345,404.593,-99.548,177.976,25.286,153.964
C04462=1090.352,404.839,-99.588,177.980,25.294,153.965
C04463=1090.358,405.086,-99.628,177.983,25.302,153.967
C04464=1090.364,405.333,-99.668,177.986,25.310,153.968
C04465=1090.370,405.580,-99.707,177.989,25.319,153.970
C04466=1090.376,405.827,-99.747,177.992,25.327,153.972
C04467=1090.383,406.073,-99.787,177.996,25.336,153.973
C04468=1090.389,406.320,-99.827,177.998,25.344,153.975
C04469=1090.395,406.567,-99.867,178.002,25.352,153.977
C04470=1090.402,406.813,-99.907,178.005,25.361,153.978
C04471=1090.407,407.061,-99.947,178.008,25.370,153.980
C04472=1090.413,407.307,-99.987,178.011,25.377,153.982
C04473=1090.420,407.554,-100.027,178.015,25.386,153.983
C04474=1090.426,407.800,-100.068,178.017,25.395,153.985
C04475=1090.433,408.047,-100.108,178.021,25.403,153.987
C04476=1090.439,408.294,-100.147,178.024,25.412,153.989
C04477=1090.444,408.541,-100.188,178.027,25.421,153.990
C04478=1090.451,408.787,-100.228,178.030,25.429,153.992
C04479=1090.457,409.034,-100.268,178.033,25.438,153.994
C04480=1090.463,409.281,-100.309,178.037,25.447,153.996
C04481=1090.469,409.527,-100.349,178.040,25.455,153.997
C04482=1090.475,409.774,-100.389,178.043,25.464,153.999
C04483=1090.482,410.020,-100.429,178.046,25.473,154.001
C04484=1090.487,410.267,-100.470,178.050,25.482,154.003
C04485=1090.494,410.513,-100.510,178.052,25.490,154.004
C04486=1090.500,410.739,-100.548,178.056,25.499,154.006
C04487=1090.505,410.964,-100.585,178.059,25.507,154.008
C04488=1090.511,411.189,-100.622,178.061,25.515,154.009
C04489=1090.516,411.414,-100.659,178.064,25.523,154.011
C04490=1090.522,411.640,-100.695,178.067,25.531,154.013
C04491=1090.528,411.865,-100.732,178.070,25.539,154.014
C04492=1090.534,412.090,-100.769,178.073,25.547,154.016
C04493=1090.540,412.316,-100.806,178.076,25.556,154.018
C04494=1090.546,412.562,-100.848,178.079,25.565,154.020
C04495=1090.552,412.808,-100.888,178.082,25.574,154.021
C04496=1090.559,413.055,-100.928,178.086,25.583,154.023
C04497=1090.564,413.302,-100.969,178.089,25.592,154.025
C04498=1090.572,413.548,-101.010,178.092,25.601,154.027
C04499=1090.577,413.795,-101.051,178.096,25.611,154.029
C04500=1090.584,414.041,-101.092,178.098,25.619,154.031
C04501=1090.590,414.288,-101.132,178.102,25.629,154.032
C04502=1090.597,414.535,-101.173,178.105,25.638,154.034
C04503=1090.603,414.781,-101.214,178.109,25.647,154.036
C04504=1090.609,415.028,-101.254,178.111,25.656,154.038
C04505=1090.616,415.274,-101.296,178.115,25.666,154.040
C04506=1090.622,415.521,-101.336,178.118,25.675,154.042
C04507=1090.629,415.767,-101.377,178.122,25.685,154.044
C04508=1090.635,416.014,-101.419,178.125,25.694,154.046
C04509=1090.641,416.261,-101.459,178.128,25.703,154.048
C04510=1090.647,416.507,-101.501,178.131,25.713,154.050
C04511=1090.654,416.754,-101.542,178.135,25.723,154.052
C04512=1090.660,417.000,-101.583,178.138,25.732,154.054
C04513=1090.666,417.246,-101.624,178.142,25.742,154.056
C04514=1090.672,417.493,-101.666,178.144,25.751,154.058
C04515=1090.679,417.740,-101.706,178.147,25.761,154.060
C04516=1090.685,417.986,-101.748,178.151,25.771,154.062
C04517=1090.691,418.232,-101.789,178.154,25.781,154.064
C04518=1090.698,418.479,-101.830,178.158,25.791,154.066
C04519=1090.704,418.725,-101.872,178.161,25.800,154.068
C04520=1090.711,418.973,-101.913,178.164,25.810,154.070
C04521=1090.717,419.219,-101.954,178.167,25.820,154.072
C04522=1090.723,419.465,-101.995,178.170,25.830,154.074
C04523=1090.730,419.712,-102.037,178.174,25.839,154.076
C04524=1090.736,419.958,-102.078,178.177,25.849,154.078
C04525=1090.742,420.205,-102.120,178.181,25.859,154.080
C04526=1090.748,420.451,-102.162,178.184,25.870,154.082
C04527=1090.755,420.698,-102.203,178.187,25.880,154.084
C04528=1090.761,420.944,-102.244,178.191,25.890,154.087
C04529=1090.768,421.189,-102.287,178.194,25.900,154.089
C04530=1090.774,421.436,-102.328,178.197,25.910,154.091
C04531=1090.780,421.682,-102.370,178.201,25.920,154.093
C04532=1090.787,421.929,-102.411,178.204,25.930,154.095
C04533=1090.794,422.176,-102.453,178.207,25.941,154.097
C04534=1090.800,422.422,-102.494,178.211,25.951,154.099
C04535=1090.807,422.668,-102.537,178.214,25.961,154.101
C04536=1090.813,422.915,-102.578,178.217,25.971,154.104
C04537=1090.819,423.162,-102.620,178.221,25.982,154.106
C04538=1090.826,423.407,-102.662,178.224,25.992,154.108
C04539=1090.832,423.654,-102.704,178.227,26.003,154.110
C04540=1090.838,423.900,-102.746,178.231,26.013,154.113
C04541=1090.845,424.146,-102.788,178.234,26.024,154.115
C04542=1090.850,424.379,-102.828,178.237,26.034,154.117
C04543=1090.857,424.612,-102.867,178.240,26.043,154.119
C04544=1090.863,424.844,-102.907,178.243,26.054,154.121
C04545=1090.869,425.077,-102.947,178.247,26.064,154.123
C04546=1090.875,425.310,-102.986,178.250,26.074,154.125
C04547=1090.881,425.543,-103.027,178.253,26.084,154.128
C04548=1090.887,425.776,-103.067,178.256,26.094,154.130
C04549=1090.893,426.008,-103.106,178.259,26.104,154.132
C04550=1090.899,426.254,-103.149,178.263,26.115,154.134
C04551=1090.906,426.501,-103.191,178.266,26.126,154.136
C04552=1090.912,426.747,-103.233,178.269,26.137,154.139
C04553=1090.919,426.993,-103.275,178.272,26.148,154.141
C04554=1090.926,427.239,-103.318,178.276,26.159,154.143
C04555=1090.932,427.485,-103.360,178.280,26.170,154.146
C04556=1090.939,427.731,-103.403,178.283,26.181,154.148
C04557=1090.945,427.979,-103.445,178.286,26.192,154.151
C04558=1090.951,428.225,-103.488,178.289,26.203,154.153
C04559=1090.958,428.470,-103.530,178.293,26.213,154.155
C04560=1090.965,428.717,-103.572,178.297,26.225,154.158
C04561=1090.971,428.963,-103.615,178.300,26.236,154.160
C04562=1090.978,429.210,-103.658,178.303,26.248,154.163
C04563=1090.984,429.455,-103.700,178.306,26.258,154.165
C04564=1090.991,429.701,-103.743,178.311,26.270,154.167
C04565=1090.997,429.948,-103.786,178.314,26.282,154.170
C04566=1091.004,430.194,-103.828,178.317,26.293,154.172
C04567=1091.010,430.440,-103.871,178.320,26.304,154.175
C04568=1091.016,430.686,-103.914,178.324,26.316,154.177
C04569=1091.023,430.932,-103.957,178.327,26.327,154.180
C04570=1091.029,431.179,-104.000,178.330,26.339,154.182
C04571=1091.036,431.425,-104.043,178.334,26.350,154.185
C04572=1091.043,431.671,-104.085,178.338,26.362,154.187
C04573=1091.049,431.917,-104.129,178.341,26.374,154.190
C04574=1091.056,432.163,-104.171,178.344,26.385,154.192
C04575=1091.062,432.409,-104.214,178.348,26.397,154.195
C04576=1091.069,432.655,-104.258,178.351,26.409,154.198
C04577=1091.075,432.902,-104.301,178.354,26.421,154.200
C04578=1091.082,433.148,-104.343,178.358,26.433,154.203
C04579=1091.088,433.394,-104.387,178.361,26.445,154.205
C04580=1091.095,433.640,-104.430,178.365,26.457,154.208
C04581=1091.102,433.886,-104.473,178.368,26.469,154.211
C04582=1091.107,434.132,-104.516,178.372,26.481,154.213
C04583=1091.114,434.378,-104.559,178.376,26.493,154.216
C04584=1091.121,434.624,-104.603,178.379,26.505,154.219
C04585=1091.127,434.870,-104.646,178.383,26.518,154.221
C04586=1091.134,435.116,-104.690,178.386,26.530,154.224
C04587=1091.140,435.362,-104.734,178.389,26.542,154.227
C04588=1091.147,435.609,-104.777,178.393,26.554,154.229
C04589=1091.154,435.854,-104.820,178.396,26.567,154.232
C04590=1091.160,436.100,-104.864,178.400,26.579,154.235
C04591=1091.167,436.346,-104.908,178.403,26.591,154.238
C04592=1091.173,436.592,-104.950,178.407,26.604,154.240
C04593=1091.180,436.838,-104.994,178.410,26.617,154.243
C04594=1091.186,437.084,-105.038,178.414,26.629,154.246
C04595=1091.193,437.330,-105.082,178.417,26.642,154.249
C04596=1091.200,437.576,-105.125,178.421,26.654,154.252
C04597=1091.206,437.822,-105.169,178.424,26.667,154.254
C04598=1091.216,438.193,-105.235,178.429,26.686,154.259
C04599=1091.227,438.563,-105.301,178.435,26.706,154.263
C04600=1091.237,438.933,-105.367,178.440,26.725,154.267
C04601=1091.247,439.304,-105.433,178.446,26.744,154.272
C04602=1091.253,439.550,-105.477,178.449,26.757,154.275
C04603=1091.260,439.796,-105.521,178.453,26.770,154.277
C04604=1091.267,440.041,-105.565,178.456,26.784,154.280
C04605=1091.274,440.287,-105.609,178.459,26.797,154.283
C04606=1091.280,440.533,-105.653,178.463,26.810,154.286
C04607=1091.287,440.779,-105.697,178.467,26.823,154.289
C04608=1091.294,441.025,-105.741,178.470,26.836,154.292
C04609=1091.300,441.271,-105.785,178.474,26.850,154.295
C04610=1091.307,441.516,-105.830,178.478,26.864,154.298
C04611=1091.314,441.763,-105.874,178.481,26.877,154.301
C04612=1091.321,442.008,-105.919,178.485,26.891,154.304
C04613=1091.327,442.254,-105.962,178.489,26.904,154.307
C04614=1091.334,442.499,-106.007,178.492,26.917,154.310
C04615=1091.341,442.746,-106.051,178.495,26.931,154.314
C04616=1091.347,442.992,-106.096,178.499,26.945,154.317
C04617=1091.354,443.237,-106.141,178.503,26.959,154.320
C04618=1091.360,443.483,-106.185,178.506,26.973,154.323
C04619=1091.368,443.729,-106.230,178.510,26.986,154.326
C04620=1091.374,443.974,-106.274,178.514,27.001,154.329
C04621=1091.382,444.220,-106.319,178.518,27.015,154.332
C04622=1091.387,444.467,-106.364,178.520,27.028,154.336
C04623=1091.394,444.712,-106.408,178.524,27.043,154.339
C04624=1091.401,444.958,-106.453,178.527,27.057,154.342
C04625=1091.408,445.203,-106.498,178.530,27.071,154.345
C04626=1091.415,445.450,-106.543,178.533,27.085,154.348
C04627=1091.421,445.695,-106.588,178.536,27.098,154.352
C04628=1091.428,445.941,-106.632,178.538,27.112,154.355
C04629=1091.435,446.187,-106.677,178.540,27.126,154.358
C04630=1091.441,446.432,-106.723,178.542,27.140,154.362
C04631=1091.449,446.678,-106.767,178.544,27.154,154.365
C04632=1091.456,446.924,-106.812,178.545,27.168,154.368
C04633=1091.462,447.170,-106.858,178.547,27.182,154.372
C04634=1091.469,447.415,-106.902,178.548,27.196,154.375
C04635=1091.476,447.661,-106.947,178.550,27.210,154.378
C04636=1091.482,447.907,-106.992,178.551,27.223,154.382
C04637=1091.490,448.153,-107.038,178.552,27.237,154.385
C04638=1091.496,448.398,-107.083,178.553,27.251,154.389
C04639=1091.503,448.644,-107.128,178.553,27.265,154.392
C04640=1091.510,448.890,-107.173,178.554,27.279,154.396
C04641=1091.516,449.136,-107.218,178.554,27.292,154.399
C04642=1091.523,449.381,-107.263,178.554,27.306,154.403
C04643=1091.531,449.627,-107.308,178.554,27.320,154.406
C04644=1091.538,449.871,-107.354,178.554,27.333,154.410
C04645=1091.547,450.118,-107.398,178.554,27.346,154.413
C04646=1091.163,450.109,-107.581,178.508,27.546,154.468
C04647=1091.153,449.863,-107.537,178.508,27.534,154.465
C04648=1091.145,449.618,-107.491,178.508,27.520,154.461
C04649=1091.139,449.372,-107.446,178.508,27.506,154.458
C04650=1091.132,449.128,-107.401,178.507,27.492,154.455
C04651=1091.125,448.881,-107.356,178.507,27.479,154.451
C04652=1091.119,448.636,-107.311,178.506,27.464,154.448
C04653=1091.111,448.390,-107.265,178.505,27.451,154.444
C04654=1091.105,448.144,-107.220,178.505,27.437,154.441
C04655=1091.098,447.899,-107.175,178.504,27.423,154.437
C04656=1091.092,447.652,-107.130,178.503,27.409,154.434
C04657=1091.085,447.408,-107.084,178.501,27.395,154.430
C04658=1091.077,447.162,-107.039,178.500,27.381,154.427
C04659=1091.071,446.915,-106.994,178.498,27.367,154.424
C04660=1091.064,446.670,-106.949,178.497,27.354,154.420
C04661=1091.057,446.424,-106.904,178.495,27.340,154.417
C04662=1091.051,446.178,-106.859,178.492,27.325,154.414
C04663=1091.043,445.932,-106.814,178.490,27.312,154.410
C04664=1091.037,445.686,-106.769,178.488,27.297,154.407
C04665=1091.031,445.441,-106.725,178.485,27.284,154.404
C04666=1091.023,445.196,-106.679,178.482,27.269,154.400
C04667=1091.016,444.950,-106.635,178.479,27.255,154.397
C04668=1091.009,444.704,-106.590,178.476,27.241,154.394
C04669=1091.003,444.458,-106.545,178.472,27.227,154.391
C04670=1090.996,444.212,-106.500,178.468,27.213,154.388
C04671=1090.989,443.966,-106.455,178.465,27.199,154.384
C04672=1090.982,443.721,-106.411,178.461,27.185,154.381
C04673=1090.975,443.475,-106.366,178.457,27.171,154.378
C04674=1090.969,443.229,-106.322,178.453,27.157,154.375
C04675=1090.963,442.983,-106.277,178.450,27.144,154.372
C04676=1090.955,442.737,-106.232,178.446,27.130,154.369
C04677=1090.949,442.492,-106.187,178.443,27.116,154.366
C04678=1090.942,442.246,-106.144,178.439,27.102,154.363
C04679=1090.935,442.000,-106.099,178.436,27.089,154.359
C04680=1090.928,441.754,-106.055,178.432,27.075,154.356
C04681=1090.922,441.509,-106.010,178.428,27.062,154.353
C04682=1090.915,441.263,-105.966,178.425,27.048,154.350
C04683=1090.908,441.017,-105.921,178.421,27.035,154.347
C04684=1090.901,440.771,-105.878,178.417,27.021,154.344
C04685=1090.895,440.525,-105.833,178.414,27.008,154.341
C04686=1090.888,440.279,-105.789,178.410,26.995,154.338
C04687=1090.881,440.033,-105.744,178.406,26.982,154.335
C04688=1090.875,439.787,-105.700,178.402,26.968,154.332
C04689=1090.868,439.541,-105.657,178.398,26.955,154.330
C04690=1090.862,439.295,-105.613,178.395,26.942,154.327
C04691=1090.851,438.937,-105.548,178.390,26.923,154.322
C04692=1090.841,438.579,-105.485,178.385,26.904,154.318
C04693=1090.832,438.221,-105.421,178.379,26.886,154.314
C04694=1090.821,437.862,-105.357,178.375,26.867,154.310
C04695=1090.815,437.616,-105.313,178.371,26.854,154.307
C04696=1090.809,437.370,-105.269,178.367,26.842,154.304
C04697=1090.801,437.125,-105.226,178.363,26.829,154.301
C04698=1090.795,436.879,-105.182,178.360,26.816,154.299
C04699=1090.789,436.633,-105.138,178.356,26.804,154.296
C04700=1090.782,436.387,-105.094,178.353,26.791,154.293
C04701=1090.775,436.141,-105.051,178.349,26.779,154.290
C04702=1090.769,435.895,-105.007,178.346,26.766,154.288
C04703=1090.762,435.649,-104.963,178.342,26.754,154.285
C04704=1090.755,435.403,-104.920,178.339,26.742,154.282
C04705=1090.749,435.157,-104.877,178.334,26.729,154.279
C04706=1090.742,434.911,-104.833,178.331,26.717,154.277
C04707=1090.735,434.665,-104.790,178.327,26.704,154.274
C04708=1090.729,434.419,-104.747,178.324,26.692,154.271
C04709=1090.723,434.173,-104.703,178.321,26.680,154.269
C04710=1090.716,433.927,-104.660,178.317,26.668,154.266
C04711=1090.709,433.680,-104.617,178.314,26.656,154.263
C04712=1090.703,433.434,-104.573,178.310,26.644,154.261
C04713=1090.696,433.188,-104.530,178.306,26.631,154.258
C04714=1090.690,432.942,-104.486,178.303,26.620,154.255
C04715=1090.683,432.696,-104.444,178.300,26.608,154.253
C04716=1090.677,432.450,-104.400,178.296,26.596,154.250
C04717=1090.670,432.204,-104.358,178.293,26.584,154.248
C04718=1090.664,431.958,-104.314,178.289,26.573,154.245
C04719=1090.657,431.712,-104.271,178.285,26.561,154.243
C04720=1090.651,431.465,-104.228,178.282,26.549,154.240
C04721=1090.644,431.220,-104.185,178.279,26.537,154.237
C04722=1090.637,430.973,-104.142,178.275,26.526,154.235
C04723=1090.631,430.727,-104.099,178.271,26.514,154.232
C04724=1090.624,430.481,-104.057,178.268,26.503,154.230
C04725=1090.618,430.235,-104.014,178.265,26.491,154.227
C04726=1090.611,429.989,-103.971,178.261,26.479,154.225
C04727=1090.604,429.743,-103.928,178.258,26.468,154.222
C04728=1090.598,429.496,-103.885,178.254,26.457,154.220
C04729=1090.592,429.251,-103.843,178.251,26.445,154.218
C04730=1090.585,429.004,-103.800,178.247,26.434,154.215
C04731=1090.579,428.758,-103.757,178.244,26.423,154.213
C04732=1090.572,428.511,-103.715,178.240,26.412,154.210
C04733=1090.565,428.265,-103.672,178.237,26.401,154.208
C04734=1090.559,428.019,-103.630,178.234,26.390,154.206
C04735=1090.553,427.773,-103.587,178.229,26.378,154.203
C04736=1090.546,427.527,-103.544,178.226,26.367,154.201
C04737=1090.539,427.280,-103.503,178.223,26.356,154.198
C04738=1090.533,427.034,-103.460,178.220,26.345,154.196
C04739=1090.526,426.788,-103.418,178.216,26.334,154.194
C04740=1090.520,426.542,-103.375,178.213,26.324,154.191
C04741=1090.513,426.296,-103.333,178.210,26.313,154.189
C04742=1090.507,426.049,-103.291,178.206,26.302,154.187
C04743=1090.501,425.816,-103.251,178.203,26.291,154.184
C04744=1090.494,425.583,-103.211,178.199,26.281,154.182
C04745=1090.488,425.350,-103.171,178.196,26.271,154.180
C04746=1090.483,425.117,-103.131,178.192,26.261,154.178
C04747=1090.476,424.883,-103.091,178.190,26.251,154.176
C04748=1090.470,424.650,-103.051,178.186,26.241,154.174
C04749=1090.465,424.416,-103.011,178.183,26.231,154.172
C04750=1090.459,424.183,-102.971,178.180,26.221,154.169
C04751=1090.452,423.937,-102.929,178.176,26.210,154.167
C04752=1090.445,423.690,-102.887,178.173,26.199,154.165
C04753=1090.439,423.445,-102.845,178.169,26.189,154.163
C04754=1090.433,423.198,-102.803,178.166,26.178,154.161
C04755=1090.427,422.951,-102.761,178.163,26.168,154.158
C04756=1090.420,422.705,-102.719,178.159,26.157,154.156
C04757=1090.414,422.459,-102.677,178.156,26.147,154.154
C04758=1090.407,422.212,-102.636,178.153,26.137,154.152
C04759=1090.401,421.966,-102.593,178.149,26.127,154.150
C04760=1090.394,421.720,-102.552,178.146,26.116,154.147
C04761=1090.388,421.474,-102.511,178.143,26.106,154.145
C04762=1090.381,421.227,-102.469,178.140,26.096,154.143
C04763=1090.375,420.981,-102.427,178.136,26.086,154.141
C04764=1090.368,420.734,-102.385,178.133,26.076,154.139
C04765=1090.362,420.488,-102.344,178.130,26.066,154.137
C04766=1090.355,420.242,-102.302,178.126,26.056,154.135
C04767=1090.349,419.995,-102.261,178.123,26.046,154.133
C04768=1090.343,419.748,-102.219,178.119,26.036,154.131
C04769=1090.337,419.502,-102.177,178.116,26.026,154.129
C04770=1090.329,419.256,-102.136,178.112,26.016,154.126
C04771=1090.323,419.009,-102.095,178.109,26.006,154.124
C04772=1090.317,418.762,-102.053,178.106,25.996,154.122
C04773=1090.311,418.516,-102.012,178.103,25.986,154.120
C04774=1090.304,418.270,-101.971,178.099,25.976,154.118
C04775=1090.298,418.023,-101.930,178.096,25.967,154.116
C04776=1090.292,417.777,-101.888,178.092,25.957,154.114
C04777=1090.286,417.530,-101.847,178.089,25.947,154.112
C04778=1090.279,417.284,-101.805,178.086,25.938,154.110
C04779=1090.273,417.038,-101.764,178.083,25.928,154.108
C04780=1090.267,416.791,-101.723,178.079,25.918,154.106
C04781=1090.260,416.544,-101.682,178.076,25.908,154.104
C04782=1090.254,416.298,-101.641,178.072,25.899,154.102
C04783=1090.248,416.051,-101.600,178.070,25.889,154.100
C04784=1090.241,415.805,-101.559,178.066,25.880,154.098
C04785=1090.235,415.558,-101.517,178.063,25.871,154.096
C04786=1090.228,415.311,-101.477,178.059,25.861,154.094
C04787=1090.222,415.065,-101.435,178.056,25.852,154.093
C04788=1090.216,414.818,-101.395,178.053,25.843,154.091
C04789=1090.209,414.572,-101.354,178.049,25.833,154.089
C04790=1090.203,414.325,-101.313,178.046,25.824,154.087
C04791=1090.196,414.079,-101.272,178.043,25.815,154.085
C04792=1090.191,413.832,-101.231,178.040,25.806,154.083
C04793=1090.183,413.586,-101.190,178.036,25.796,154.081
C04794=1090.178,413.339,-101.149,178.033,25.787,154.079
C04795=1090.171,413.092,-101.109,178.030,25.778,154.077
C04796=1090.165,412.847,-101.068,178.026,25.769,154.076
C04797=1090.158,412.599,-101.027,178.023,25.760,154.074
C04798=1090.152,412.352,-100.987,178.020,25.751,154.072
C04799=1090.146,412.127,-100.950,178.017,25.742,154.070
C04800=1090.140,411.902,-100.913,178.014,25.734,154.068
C04801=1090.135,411.676,-100.875,178.011,25.726,154.067
C04802=1090.129,411.449,-100.838,178.008,25.717,154.065
C04803=1090.124,411.224,-100.801,178.005,25.709,154.063
C04804=1090.118,410.999,-100.764,178.002,25.701,154.062
C04805=1090.112,410.772,-100.727,177.999,25.693,154.060
C04806=1090.106,410.547,-100.690,177.996,25.685,154.059
C04807=1090.100,410.301,-100.650,177.993,25.676,154.057
C04808=1090.094,410.053,-100.609,177.989,25.667,154.055
C04809=1090.087,409.807,-100.569,177.986,25.658,154.053
C04810=1090.081,409.560,-100.528,177.983,25.650,154.051
C04811=1090.075,409.314,-100.488,177.980,25.641,154.050
C04812=1090.069,409.067,-100.448,177.977,25.632,154.048
C04813=1090.063,408.821,-100.407,177.974,25.624,154.046
C04814=1090.056,408.574,-100.367,177.970,25.614,154.044
C04815=1090.051,408.327,-100.326,177.967,25.606,154.043
C04816=1090.044,408.081,-100.286,177.964,25.597,154.041
C04817=1090.038,407.834,-100.246,177.961,25.589,154.039
C04818=1090.031,407.588,-100.206,177.957,25.580,154.037
C04819=1090.026,407.340,-100.166,177.955,25.572,154.036
C04820=1090.020,407.094,-100.126,177.951,25.563,154.034
C04821=1090.013,406.847,-100.086,177.948,25.555,154.032
C04822=1090.007,406.601,-100.046,177.945,25.546,154.031
C04823=1090.001,406.354,-100.005,177.942,25.538,154.029
C04824=1089.995,406.107,-99.966,177.938,25.529,154.027
C04825=1089.988,405.860,-99.926,177.935,25.521,154.026
C04826=1089.982,405.614,-99.886,177.932,25.512,154.024
C04827=1089.976,405.367,-99.846,177.929,25.504,154.022
C04828=1089.969,405.120,-99.806,177.925,25.496,154.021
C04829=1089.963,404.874,-99.766,177.922,25.487,154.019
C04830=1089.957,404.627,-99.727,177.920,25.479,154.017
C04831=1089.950,404.380,-99.686,177.916,25.471,154.016
C04832=1089.944,404.133,-99.647,177.913,25.463,154.014
C04833=1089.938,403.886,-99.607,177.909,25.454,154.012
C04834=1089.932,403.639,-99.567,177.906,25.446,154.011
C04835=1089.926,403.394,-99.528,177.904,25.438,154.009
C04836=1089.920,403.146,-99.488,177.900,25.430,154.008
C04837=1089.914,402.900,-99.448,177.897,25.422,154.006
C04838=1089.908,402.653,-99.409,177.893,25.414,154.005
C04839=1089.902,402.406,-99.369,177.890,25.406,154.003
C04840=1089.895,402.159,-99.329,177.888,25.398,154.001
C04841=1089.888,401.912,-99.290,177.884,25.390,154.000
C04842=1089.882,401.665,-99.251,177.881,25.382,153.998
C04843=1089.877,401.419,-99.211,177.878,25.374,153.997
C04844=1089.870,401.172,-99.172,177.874,25.366,153.995
C04845=1089.864,400.925,-99.132,177.872,25.358,153.994
C04846=1089.858,400.678,-99.093,177.869,25.351,153.992
C04847=1089.851,400.432,-99.053,177.865,25.342,153.991
C04848=1089.846,400.185,-99.014,177.862,25.335,153.989
C04849=1089.840,399.938,-98.975,177.859,25.327,153.987
C04850=1089.834,399.691,-98.935,177.856,25.319,153.986
C04851=1089.827,399.444,-98.896,177.852,25.311,153.985
C04852=1089.821,399.198,-98.857,177.849,25.304,153.983
C04853=1089.815,398.951,-98.818,177.847,25.296,153.981
C04854=1089.809,398.703,-98.778,177.843,25.288,153.980
C04855=1089.803,398.478,-98.743,177.841,25.281,153.979
C04856=1089.798,398.254,-98.707,177.838,25.274,153.977
C04857=1089.792,398.028,-98.672,177.835,25.267,153.976
C04858=1089.786,397.803,-98.636,177.832,25.260,153.975
C04859=1089.780,397.578,-98.600,177.829,25.253,153.973
C04860=1089.776,397.353,-98.564,177.826,25.247,153.972
C04861=1089.770,397.128,-98.529,177.823,25.240,153.971
C04862=1089.764,396.902,-98.493,177.820,25.233,153.969
C04863=1089.757,396.656,-98.454,177.817,25.225,153.968
C04864=1089.751,396.409,-98.415,177.814,25.217,153.966
C04865=1089.745,396.162,-98.376,177.811,25.210,153.965
C04866=1089.739,395.916,-98.337,177.807,25.202,153.964
C04867=1089.733,395.668,-98.298,177.805,25.195,153.962
C04868=1089.727,395.422,-98.260,177.802,25.188,153.961
C04869=1089.721,395.175,-98.220,177.799,25.180,153.959
C04870=1089.714,394.928,-98.182,177.796,25.173,153.958
C04871=1089.709,394.681,-98.143,177.792,25.165,153.957
C04872=1089.702,394.434,-98.104,177.789,25.158,153.955
C04873=1089.697,394.188,-98.065,177.786,25.151,153.954
C04874=1089.690,393.940,-98.027,177.783,25.144,153.952
C04875=1089.684,393.693,-97.988,177.780,25.136,153.951
C04876=1089.678,393.447,-97.949,177.777,25.129,153.950
C04877=1089.671,393.199,-97.911,177.773,25.122,153.948
C04878=1089.666,392.953,-97.872,177.770,25.115,153.947
C04879=1089.659,392.706,-97.833,177.767,25.108,153.946
C04880=1089.654,392.459,-97.795,177.764,25.100,153.944
C04881=1089.647,392.212,-97.756,177.761,25.093,153.943
C04882=1089.641,391.966,-97.718,177.758,25.086,153.942
C04883=1089.635,391.718,-97.679,177.755,25.079,153.940
C04884=1089.629,391.472,-97.641,177.751,25.072,153.939
C04885=1089.623,391.225,-97.602,177.748,25.065,153.938
C04886=1089.617,390.978,-97.565,177.745,25.058,153.936
C04887=1089.610,390.731,-97.526,177.742,25.051,153.935
C04888=1089.605,390.484,-97.487,177.739,25.044,153.934
C04889=1089.598,390.237,-97.449,177.736,25.037,153.932
C04890=1089.592,389.991,-97.411,177.733,25.030,153.931
C04891=1089.585,389.743,-97.373,177.730,25.023,153.930
C04892=1089.580,389.496,-97.335,177.727,25.016,153.929
C04893=1089.573,389.250,-97.296,177.723,25.009,153.927
C04894=1089.567,389.003,-97.258,177.719,25.002,153.926
C04895=1089.562,388.756,-97.220,177.717,24.995,153.925
C04896=1089.555,388.508,-97.182,177.713,24.988,153.924
C04897=1089.549,388.262,-97.143,177.710,24.982,153.922
C04898=1089.543,388.016,-97.106,177.707,24.975,153.921
C04899=1089.537,387.768,-97.068,177.704,24.968,153.920
C04900=1089.531,387.521,-97.030,177.701,24.961,153.919
C04901=1089.525,387.275,-96.992,177.698,24.955,153.917
C04902=1089.518,387.027,-96.954,177.695,24.948,153.916
C04903=1089.512,386.780,-96.916,177.692,24.941,153.915
C04904=1089.507,386.534,-96.877,177.689,24.934,153.914
C04905=1089.500,386.287,-96.839,177.686,24.928,153.912
C04906=1089.494,386.040,-96.801,177.682,24.921,153.911
C04907=1089.488,385.793,-96.763,177.679,24.914,153.910
C04908=1089.482,385.546,-96.725,177.676,24.908,153.909
C04909=1089.476,385.299,-96.688,177.673,24.901,153.908
C04910=1089.470,385.052,-96.650,177.670,24.894,153.906
C04911=1089.465,384.833,-96.617,177.667,24.888,153.905
C04912=1089.460,384.614,-96.583,177.664,24.882,153.904
C04913=1089.454,384.396,-96.550,177.661,24.877,153.903
C04914=1089.449,384.177,-96.516,177.659,24.871,153.902
C04915=1089.444,383.959,-96.483,177.656,24.865,153.901
C04916=1089.439,383.740,-96.449,177.653,24.859,153.900
C04917=1089.433,383.522,-96.416,177.651,24.853,153.899
C04918=1089.428,383.304,-96.383,177.647,24.847,153.898
C04919=1089.421,383.057,-96.345,177.644,24.841,153.897
C04920=1089.415,382.810,-96.307,177.641,24.834,153.896
C04921=1089.410,382.563,-96.270,177.638,24.828,153.894
C04922=1089.404,382.316,-96.233,177.635,24.821,153.893
C04923=1089.397,382.069,-96.195,177.632,24.815,153.892
C04924=1089.392,381.821,-96.158,177.629,24.809,153.891
C04925=1089.386,381.575,-96.120,177.625,24.802,153.890
C04926=1089.379,381.328,-96.083,177.623,24.796,153.889
C04927=1089.374,381.081,-96.046,177.620,24.790,153.888
C04928=1089.367,380.833,-96.007,177.617,24.784,153.887
C04929=1089.361,380.587,-95.970,177.613,24.777,153.886
C04930=1089.355,380.340,-95.933,177.610,24.771,153.884
C04931=1089.349,380.093,-95.895,177.607,24.765,153.883
C04932=1089.343,379.845,-95.858,177.604,24.758,153.882
C04933=1089.337,379.599,-95.821,177.601,24.752,153.881
C04934=1089.331,379.351,-95.784,177.598,24.746,153.880
C04935=1089.325,379.104,-95.746,177.594,24.740,153.879
C04936=1089.319,378.857,-95.709,177.591,24.733,153.878
C04937=1089.312,378.610,-95.672,177.588,24.727,153.877
C04938=1089.307,378.363,-95.635,177.586,24.721,153.876
C04939=1089.301,378.116,-95.598,177.582,24.715,153.875
C04940=1089.295,377.869,-95.561,177.579,24.709,153.874
C04941=1089.289,377.622,-95.524,177.576,24.703,153.872
C04942=1089.283,377.375,-95.486,177.573,24.696,153.871
C04943=1089.277,377.128,-95.449,177.570,24.690,153.870
C04944=1089.271,376.881,-95.412,177.566,24.684,153.869
C04945=1089.266,376.633,-95.375,177.563,24.678,153.868
C04946=1089.259,376.387,-95.338,177.560,24.672,153.867
C04947=1089.253,376.139,-95.301,177.557,24.666,153.866
C04948=1089.247,375.891,-95.264,177.554,24.660,153.865
C04949=1089.241,375.644,-95.227,177.551,24.654,153.864
C04950=1089.235,375.398,-95.190,177.548,24.648,153.863
C04951=1089.229,375.151,-95.153,177.545,24.642,153.862
C04952=1089.224,374.904,-95.116,177.541,24.635,153.861
C04953=1089.218,374.657,-95.079,177.539,24.630,153.860
C04954=1089.212,374.410,-95.043,177.536,24.624,153.859
C04955=1089.206,374.162,-95.006,177.532,24.618,153.858
C04956=1089.200,373.915,-94.969,177.529,24.612,153.857
C04957=1089.194,373.668,-94.932,177.526,24.606,153.856
C04958=1089.188,373.421,-94.896,177.523,24.600,153.855
C04959=1089.181,373.174,-94.860,177.520,24.594,153.854
C04960=1089.176,372.926,-94.822,177.517,24.589,153.853
C04961=1089.169,372.679,-94.786,177.514,24.583,153.852
C04962=1089.163,372.432,-94.750,177.510,24.577,153.851
C04963=1089.158,372.185,-94.713,177.507,24.571,153.850
C04964=1089.151,371.938,-94.676,177.505,24.565,153.849
C04965=1089.146,371.690,-94.639,177.501,24.560,153.848
C04966=1089.139,371.443,-94.603,177.498,24.554,153.847
C04967=1089.129,371.033,-94.542,177.493,24.544,153.845
C04968=1089.120,370.625,-94.481,177.488,24.535,153.844
C04969=1089.109,370.216,-94.422,177.482,24.525,153.842
C04970=1089.100,369.807,-94.361,177.477,24.515,153.841
C04971=1089.094,369.559,-94.326,177.475,24.511,153.840
C04972=1089.088,369.312,-94.288,177.471,24.505,153.839
C04973=1089.082,369.065,-94.252,177.468,24.499,153.838
C04974=1089.076,368.817,-94.216,177.465,24.493,153.837
C04975=1089.069,368.570,-94.180,177.462,24.488,153.836
C04976=1089.064,368.323,-94.143,177.459,24.482,153.835
C04977=1089.058,368.076,-94.107,177.456,24.476,153.834
C04978=1089.052,367.829,-94.071,177.452,24.470,153.833
C04979=1089.046,367.581,-94.034,177.450,24.465,153.832
C04980=1089.040,367.334,-93.998,177.447,24.460,153.831
C04981=1089.034,367.087,-93.962,177.443,24.454,153.830
C04982=1089.029,366.840,-93.926,177.440,24.448,153.829
C04983=1089.022,366.593,-93.890,177.437,24.443,153.829
C04984=1089.017,366.345,-93.854,177.434,24.437,153.828
C04985=1089.011,366.097,-93.817,177.431,24.431,153.827
C04986=1089.005,365.851,-93.782,177.428,24.427,153.826
C04987=1088.999,365.603,-93.745,177.425,24.421,153.825
C04988=1088.993,365.356,-93.710,177.421,24.415,153.824
C04989=1088.987,365.108,-93.674,177.418,24.410,153.823
C04990=1088.980,364.861,-93.638,177.416,24.405,153.822
C04991=1088.976,364.614,-93.602,177.412,24.399,153.821
C04992=1088.970,364.366,-93.566,177.409,24.393,153.820
C04993=1088.963,364.119,-93.529,177.406,24.389,153.820
C04994=1088.957,363.871,-93.494,177.403,24.383,153.819
C04995=1088.952,363.624,-93.458,177.400,24.377,153.818
C04996=1088.946,363.377,-93.422,177.397,24.372,153.817
C04997=1088.940,363.130,-93.386,177.394,24.367,153.816
C04998=1088.933,362.882,-93.350,177.390,24.361,153.815
C04999=1088.928,362.635,-93.315,177.388,24.356,153.814
C05000=1088.921,362.388,-93.280,177.384,24.351,153.814
C05001=1088.915,362.141,-93.243,177.381,24.345,153.813
C05002=1088.910,361.894,-93.208,177.379,24.340,153.812
C05003=1088.904,361.646,-93.172,177.375,24.335,153.811
C05004=1088.897,361.398,-93.137,177.372,24.330,153.810
C05005=1088.892,361.151,-93.101,177.369,24.325,153.809
C05006=1088.886,360.904,-93.066,177.366,24.319,153.809
C05007=1088.880,360.656,-93.030,177.362,24.314,153.808
C05008=1088.875,360.409,-92.994,177.360,24.309,153.807
C05009=1088.869,360.161,-92.959,177.356,24.304,153.806
C05010=1088.862,359.914,-92.923,177.353,24.298,153.805
C05011=1088.857,359.667,-92.888,177.350,24.293,153.804
C05012=1088.850,359.419,-92.852,177.347,24.288,153.804
C05013=1088.844,359.172,-92.817,177.344,24.283,153.803
C05014=1088.839,358.925,-92.781,177.341,24.278,153.802
C05015=1088.833,358.677,-92.746,177.338,24.272,153.801
C05016=1088.826,358.430,-92.711,177.335,24.268,153.801
C05017=1088.821,358.183,-92.675,177.331,24.262,153.800
C05018=1088.815,357.935,-92.639,177.328,24.257,153.799
C05019=1088.806,357.541,-92.583,177.323,24.249,153.798
C05020=1088.795,357.148,-92.527,177.319,24.241,153.796
C05021=1088.786,356.754,-92.471,177.313,24.233,153.795
C05022=1088.777,356.361,-92.415,177.309,24.225,153.794
C05023=1088.772,356.112,-92.380,177.306,24.220,153.793
C05024=1088.765,355.865,-92.345,177.303,24.215,153.792
C05025=1088.760,355.618,-92.310,177.299,24.209,153.792
C05026=1088.753,355.370,-92.274,177.296,24.205,153.791
C05027=1088.748,355.123,-92.240,177.293,24.200,153.790
C05028=1088.742,354.875,-92.204,177.290,24.195,153.789
C05029=1088.736,354.628,-92.169,177.287,24.190,153.788
C05030=1088.730,354.380,-92.134,177.284,24.185,153.788
C05031=1088.724,354.133,-92.099,177.281,24.180,153.787
C05032=1088.719,353.885,-92.064,177.277,24.175,153.786
C05033=1088.712,353.638,-92.029,177.275,24.170,153.785
C05034=1088.707,353.390,-91.994,177.271,24.165,153.785
C05035=1088.700,353.144,-91.959,177.269,24.160,153.784
C05036=1088.695,352.896,-91.925,177.265,24.155,153.783
C05037=1088.689,352.648,-91.889,177.263,24.150,153.782
C05038=1088.683,352.401,-91.855,177.259,24.145,153.782
C05039=1088.677,352.153,-91.819,177.256,24.141,153.781
C05040=1088.672,351.906,-91.785,177.253,24.136,153.780
C05041=1088.665,351.659,-91.750,177.250,24.131,153.780
C05042=1088.660,351.411,-91.715,177.247,24.126,153.779
C05043=1088.653,351.163,-91.681,177.243,24.121,153.778
C05044=1088.648,350.916,-91.646,177.241,24.117,153.777
C05045=1088.641,350.668,-91.611,177.237,24.112,153.777
C05046=1088.636,350.421,-91.577,177.235,24.107,153.776
C05047=1088.630,350.174,-91.542,177.231,24.102,153.775
C05048=1088.624,349.926,-91.507,177.228,24.097,153.775
C05049=1088.618,349.678,-91.473,177.225,24.092,153.774
C05050=1088.612,349.430,-91.438,177.222,24.088,153.773
C05051=1088.607,349.183,-91.403,177.219,24.083,153.773
C05052=1088.601,348.936,-91.369,177.216,24.078,153.772
C05053=1088.595,348.688,-91.334,177.212,24.074,153.771
C05054=1088.589,348.440,-91.300,177.210,24.069,153.770
C05055=1088.583,348.193,-91.266,177.206,24.064,153.770
C05056=1088.577,347.946,-91.230,177.204,24.060,153.769
C05057=1088.571,347.698,-91.196,177.200,24.055,153.768
C05058=1088.565,347.450,-91.162,177.197,24.050,153.768
C05059=1088.560,347.203,-91.127,177.194,24.045,153.767
C05060=1088.554,346.955,-91.093,177.191,24.041,153.766
C05061=1088.548,346.708,-91.059,177.189,24.036,153.766
C05062=1088.542,346.460,-91.024,177.185,24.031,153.765
C05063=1088.536,346.212,-90.990,177.182,24.027,153.764
C05064=1088.531,345.965,-90.956,177.179,24.022,153.764
C05065=1088.525,345.717,-90.921,177.176,24.017,153.763
C05066=1088.519,345.470,-90.887,177.173,24.013,153.762
C05067=1088.513,345.222,-90.853,177.170,24.008,153.762
C05068=1088.507,344.975,-90.819,177.166,24.003,153.761
C05069=1088.502,344.727,-90.784,177.164,23.999,153.760
C05070=1088.496,344.479,-90.749,177.160,23.994,153.760
C05071=1088.486,344.088,-90.696,177.155,23.987,153.759
C05072=1088.477,343.698,-90.642,177.150,23.980,153.758
C05073=1088.468,343.306,-90.588,177.145,23.973,153.757
C05074=1088.458,342.915,-90.534,177.141,23.966,153.756
C05075=1088.452,342.668,-90.500,177.138,23.961,153.755
C05076=1088.446,342.421,-90.466,177.135,23.957,153.754
C05077=1088.441,342.173,-90.433,177.132,23.952,153.754
C05078=1088.436,341.925,-90.398,177.129,23.948,153.753
C05079=1088.429,341.677,-90.364,177.125,23.943,153.752
C05080=1088.423,341.430,-90.330,177.123,23.939,153.752
C05081=1088.418,341.182,-90.296,177.120,23.935,153.751
C05082=1088.412,340.935,-90.262,177.116,23.930,153.751
C05083=1088.406,340.687,-90.228,177.114,23.926,153.750
C05084=1088.400,340.439,-90.195,177.110,23.921,153.749
C05085=1088.394,340.191,-90.161,177.107,23.917,153.749
C05086=1088.388,339.944,-90.127,177.105,23.913,153.748
C05087=1088.382,339.696,-90.093,177.101,23.908,153.747
C05088=1088.377,339.449,-90.059,177.098,23.904,153.747
C05089=1088.371,339.201,-90.026,177.095,23.899,153.746
C05090=1088.365,338.954,-89.992,177.092,23.895,153.746
C05091=1088.359,338.705,-89.958,177.089,23.891,153.745
C05092=1088.353,338.458,-89.924,177.086,23.886,153.744
C05093=1088.348,338.210,-89.891,177.083,23.882,153.744
C05094=1088.342,337.963,-89.857,177.080,23.877,153.743
C05095=1088.336,337.715,-89.823,177.077,23.873,153.743
C05096=1088.330,337.467,-89.790,177.074,23.868,153.742
C05097=1088.324,337.220,-89.756,177.070,23.864,153.741
C05098=1088.319,336.972,-89.723,177.067,23.860,153.741
C05099=1088.312,336.724,-89.689,177.065,23.856,153.740
C05100=1088.306,336.476,-89.655,177.061,23.851,153.740
C05101=1088.301,336.228,-89.622,177.058,23.847,153.739
C05102=1088.294,335.981,-89.588,177.055,23.843,153.738
C05103=1088.289,335.733,-89.555,177.052,23.838,153.738
C05104=1088.283,335.485,-89.522,177.049,23.834,153.737
C05105=1088.277,335.238,-89.488,177.046,23.830,153.737
C05106=1088.272,334.990,-89.454,177.043,23.826,153.736
C05107=1088.266,334.743,-89.422,177.040,23.822,153.736
C05108=1088.260,334.495,-89.388,177.037,23.817,153.735
C05109=1088.254,334.247,-89.355,177.034,23.813,153.734
C05110=1088.249,334.000,-89.321,177.031,23.809,153.734
C05111=1088.243,333.752,-89.288,177.028,23.804,153.733
C05112=1088.237,333.504,-89.255,177.024,23.800,153.733
C05113=1088.231,333.256,-89.222,177.022,23.796,153.732
C05114=1088.226,333.008,-89.188,177.019,23.792,153.732
C05115=1088.219,332.761,-89.155,177.016,23.788,153.731
C05116=1088.213,332.513,-89.121,177.012,23.783,153.731
C05117=1088.208,332.265,-89.088,177.010,23.779,153.730
C05118=1088.202,332.018,-89.055,177.007,23.775,153.729
C05119=1088.196,331.770,-89.022,177.003,23.771,153.729
C05120=1088.190,331.522,-88.989,177.000,23.767,153.728
C05121=1088.184,331.274,-88.956,176.997,23.763,153.728
C05122=1088.179,331.027,-88.923,176.994,23.758,153.727
C05123=1088.168,330.630,-88.870,176.990,23.752,153.726
C05124=1088.159,330.233,-88.817,176.985,23.746,153.726
C05125=1088.150,329.836,-88.764,176.980,23.739,153.725
C05126=1088.140,329.440,-88.712,176.975,23.733,153.724
C05127=1088.134,329.192,-88.678,176.972,23.729,153.723
C05128=1088.128,328.944,-88.646,176.969,23.725,153.723
C05129=1088.123,328.696,-88.613,176.965,23.721,153.723
C05130=1088.117,328.448,-88.580,176.962,23.717,153.722
C05131=1088.110,328.200,-88.547,176.960,23.712,153.721
C05132=1088.105,327.953,-88.514,176.957,23.709,153.721
C05133=1088.098,327.705,-88.481,176.953,23.704,153.720
C05134=1088.093,327.456,-88.449,176.950,23.701,153.720
C05135=1088.088,327.210,-88.416,176.947,23.697,153.719
C05136=1088.081,326.962,-88.384,176.945,23.693,153.719
C05137=1088.076,326.714,-88.350,176.941,23.689,153.718
C05138=1088.070,326.466,-88.318,176.938,23.684,153.718
C05139=1088.064,326.218,-88.285,176.935,23.681,153.717
C05140=1088.058,325.970,-88.252,176.932,23.677,153.717
C05141=1088.052,325.722,-88.220,176.929,23.672,153.716
C05142=1088.047,325.475,-88.187,176.926,23.669,153.716
C05143=1088.041,325.227,-88.154,176.923,23.665,153.715
C05144=1088.035,324.979,-88.122,176.920,23.661,153.715
C05145=1088.029,324.731,-88.089,176.917,23.657,153.714
C05146=1088.023,324.483,-88.057,176.914,23.653,153.714
C05147=1088.017,324.235,-88.024,176.911,23.649,153.713
C05148=1088.012,323.988,-87.992,176.908,23.645,153.713
C05149=1088.006,323.740,-87.959,176.905,23.641,153.712
C05150=1088.000,323.492,-87.927,176.901,23.637,153.712
C05151=1087.994,323.244,-87.895,176.899,23.633,153.711
C05152=1087.989,322.997,-87.862,176.896,23.629,153.711
C05153=1087.983,322.749,-87.830,176.893,23.625,153.710
C05154=1087.977,322.501,-87.798,176.890,23.622,153.710
C05155=1087.971,322.253,-87.764,176.887,23.618,153.709
C05156=1087.966,322.005,-87.733,176.883,23.614,153.709
C05157=1087.959,321.758,-87.700,176.881,23.610,153.709
C05158=1087.953,321.509,-87.668,176.878,23.606,153.708
C05159=1087.949,321.262,-87.635,176.875,23.602,153.708
C05160=1087.943,321.014,-87.603,176.872,23.598,153.707
C05161=1087.937,320.766,-87.571,176.868,23.594,153.707
C05162=1087.930,320.518,-87.538,176.866,23.590,153.706
C05163=1087.926,320.270,-87.506,176.863,23.586,153.706
C05164=1087.920,320.022,-87.474,176.860,23.583,153.705
C05165=1087.914,319.775,-87.441,176.857,23.579,153.705
C05166=1087.908,319.527,-87.409,176.854,23.575,153.704
C05167=1087.902,319.279,-87.377,176.850,23.571,153.704
C05168=1087.897,319.031,-87.345,176.848,23.567,153.703
C05169=1087.891,318.783,-87.312,176.845,23.563,153.703
C05170=1087.885,318.535,-87.280,176.842,23.559,153.702
C05171=1087.880,318.288,-87.249,176.839,23.556,153.702
C05172=1087.874,318.039,-87.217,176.836,23.552,153.701
C05173=1087.868,317.792,-87.185,176.833,23.547,153.701
C05174=1087.863,317.543,-87.152,176.830,23.544,153.700
C05175=1087.853,317.140,-87.100,176.825,23.538,153.700
C05176=1087.844,316.736,-87.048,176.820,23.532,153.699
C05177=1087.835,316.332,-86.995,176.815,23.525,153.698
C05178=1087.826,315.930,-86.944,176.810,23.519,153.697
C05179=1087.820,315.682,-86.912,176.807,23.515,153.697
C05180=1087.815,315.434,-86.880,176.804,23.512,153.697
C05181=1087.809,315.186,-86.848,176.802,23.508,153.696
C05182=1087.804,314.938,-86.816,176.799,23.504,153.696
C05183=1087.797,314.690,-86.785,176.796,23.500,153.695
C05184=1087.791,314.442,-86.752,176.793,23.497,153.695
C05185=1087.786,314.194,-86.721,176.790,23.493,153.694
C05186=1087.780,313.946,-86.689,176.786,23.489,153.694
C05187=1087.773,313.698,-86.657,176.783,23.485,153.694
C05188=1087.768,313.451,-86.626,176.780,23.482,153.693
C05189=1087.762,313.202,-86.594,176.777,23.479,153.693
C05190=1087.757,312.954,-86.563,176.774,23.475,153.692
C05191=1087.750,312.707,-86.531,176.772,23.471,153.692
C05192=1087.745,312.459,-86.500,176.769,23.468,153.692
C05193=1087.739,312.211,-86.468,176.766,23.464,153.691
C05194=1087.732,311.964,-86.437,176.763,23.460,153.691
C05195=1087.727,311.715,-86.405,176.759,23.456,153.690
C05196=1087.721,311.467,-86.373,176.756,23.453,153.690
C05197=1087.715,311.219,-86.342,176.753,23.450,153.690
C05198=1087.709,310.971,-86.310,176.750,23.446,153.689
C05199=1087.703,310.724,-86.278,176.747,23.442,153.689
C05200=1087.698,310.475,-86.247,176.744,23.439,153.688
C05201=1087.692,310.228,-86.216,176.742,23.435,153.688
C05202=1087.686,309.980,-86.184,176.739,23.431,153.687
C05203=1087.680,309.731,-86.153,176.736,23.428,153.687
C05204=1087.674,309.484,-86.122,176.733,23.425,153.687
C05205=1087.668,309.236,-86.090,176.730,23.421,153.686
C05206=1087.663,308.988,-86.059,176.726,23.417,153.686
C05207=1087.657,308.740,-86.028,176.723,23.413,153.685
C05208=1087.651,308.492,-85.996,176.720,23.410,153.685
C05209=1087.645,308.244,-85.966,176.717,23.407,153.685
C05210=1087.639,307.996,-85.934,176.714,23.403,153.684
C05211=1087.634,307.748,-85.903,176.711,23.399,153.684
C05212=1087.628,307.500,-85.871,176.709,23.396,153.683
C05213=1087.622,307.252,-85.840,176.706,23.392,153.683
C05214=1087.616,307.005,-85.809,176.703,23.389,153.683
C05215=1087.611,306.756,-85.778,176.700,23.385,153.682
C05216=1087.605,306.509,-85.746,176.697,23.382,153.682
C05217=1087.599,306.261,-85.716,176.694,23.378,153.681
C05218=1087.593,306.013,-85.684,176.691,23.374,153.681
C05219=1087.588,305.765,-85.653,176.688,23.371,153.681
C05220=1087.582,305.517,-85.622,176.684,23.367,153.680
C05221=1087.576,305.269,-85.591,176.681,23.363,153.680
C05222=1087.570,305.021,-85.559,176.678,23.360,153.680
C05223=1087.565,304.773,-85.529,176.675,23.357,153.679
C05224=1087.560,304.525,-85.498,176.672,23.353,153.679
C05225=1087.554,304.277,-85.466,176.670,23.349,153.678
C05226=1087.548,304.029,-85.436,176.667,23.346,153.678
C05227=1087.539,303.628,-85.386,176.662,23.340,153.677
C05228=1087.530,303.228,-85.336,176.657,23.334,153.677
C05229=1087.521,302.827,-85.286,176.653,23.329,153.676
C05230=1087.511,302.426,-85.236,176.648,23.323,153.675
C05231=1087.505,302.178,-85.204,176.645,23.320,153.675
C05232=1087.500,301.930,-85.174,176.642,23.316,153.675
C05233=1087.495,301.682,-85.143,176.639,23.313,153.674
C05234=1087.489,301.434,-85.113,176.636,23.309,153.674
C05235=1087.484,301.186,-85.082,176.633,23.306,153.674
C05236=1087.477,300.937,-85.051,176.630,23.302,153.673
C05237=1087.471,300.690,-85.020,176.627,23.299,153.673
C05238=1087.466,300.442,-84.989,176.624,23.295,153.672
C05239=1087.460,300.194,-84.959,176.621,23.292,153.672
C05240=1087.455,299.946,-84.928,176.618,23.288,153.672
C05241=1087.449,299.698,-84.897,176.615,23.285,153.671
C05242=1087.444,299.450,-84.866,176.612,23.281,153.671
C05243=1087.438,299.202,-84.836,176.610,23.277,153.671
C05244=1087.432,298.954,-84.805,176.606,23.274,153.670
C05245=1087.427,298.706,-84.774,176.604,23.271,153.670
C05246=1087.421,298.458,-84.744,176.601,23.267,153.669
C05247=1087.416,298.210,-84.713,176.598,23.264,153.669
C05248=1087.410,297.962,-84.683,176.595,23.260,153.669
C05249=1087.404,297.714,-84.652,176.592,23.257,153.668
C05250=1087.399,297.466,-84.622,176.589,23.253,153.668
C05251=1087.393,297.217,-84.591,176.586,23.250,153.668
C05252=1087.387,296.970,-84.560,176.583,23.247,153.667
C05253=1087.381,296.722,-84.530,176.580,23.243,153.667
C05254=1087.375,296.474,-84.500,176.577,23.240,153.667
C05255=1087.370,296.226,-84.469,176.574,23.237,153.666
C05256=1087.365,295.977,-84.439,176.571,23.233,153.666
C05257=1087.359,295.730,-84.409,176.568,23.230,153.666
C05258=1087.353,295.482,-84.378,176.565,23.227,153.665
C05259=1087.347,295.233,-84.348,176.562,23.223,153.665
C05260=1087.341,294.985,-84.317,176.559,23.220,153.665
C05261=1087.335,294.737,-84.288,176.556,23.217,153.664
C05262=1087.330,294.489,-84.257,176.553,23.213,153.664
C05263=1087.324,294.241,-84.227,176.550,23.210,153.664
C05264=1087.318,293.993,-84.197,176.547,23.206,153.663
C05265=1087.312,293.745,-84.167,176.544,23.203,153.663
C05266=1087.307,293.497,-84.137,176.541,23.200,153.663
C05267=1087.302,293.249,-84.106,176.538,23.196,153.662
C05268=1087.296,293.001,-84.076,176.536,23.193,153.662
C05269=1087.290,292.753,-84.046,176.533,23.190,153.662
C05270=1087.284,292.505,-84.015,176.530,23.186,153.661
C05271=1087.279,292.257,-83.986,176.527,23.183,153.661
C05272=1087.273,292.009,-83.955,176.524,23.180,153.660
C05273=1087.267,291.761,-83.925,176.521,23.176,153.660
C05274=1087.262,291.512,-83.895,176.518,23.173,153.660
C05275=1087.255,291.264,-83.865,176.515,23.170,153.659
C05276=1087.250,291.015,-83.835,176.512,23.166,153.659
C05277=1087.244,290.768,-83.805,176.509,23.163,153.659
C05278=1087.239,290.519,-83.775,176.506,23.160,153.659
C05279=1087.230,290.133,-83.728,176.502,23.155,153.658
C05280=1087.220,289.746,-83.682,176.498,23.150,153.657
C05281=1087.211,289.360,-83.635,176.493,23.145,153.657
C05282=1087.203,288.973,-83.589,176.489,23.140,153.656
C05283=1087.197,288.726,-83.559,176.486,23.136,153.656
C05284=1087.191,288.477,-83.529,176.483,23.133,153.656
C05285=1087.186,288.229,-83.500,176.480,23.130,153.656
C05286=1087.180,287.981,-83.469,176.477,23.126,153.655
C05287=1087.174,287.732,-83.440,176.474,23.123,153.655
C05288=1087.168,287.484,-83.410,176.471,23.120,153.655
C05289=1087.162,287.236,-83.380,176.468,23.117,153.654
C05290=1087.157,286.988,-83.351,176.465,23.114,153.654
C05291=1087.151,286.740,-83.321,176.462,23.111,153.654
C05292=1087.145,286.492,-83.291,176.460,23.107,153.653
C05293=1087.139,286.244,-83.261,176.456,23.104,153.653
C05294=1087.134,285.995,-83.232,176.453,23.101,153.653
C05295=1087.128,285.747,-83.202,176.450,23.098,153.652
C05296=1087.122,285.499,-83.172,176.447,23.094,153.652
C05297=1087.117,285.251,-83.143,176.445,23.091,153.652
C05298=1087.111,285.003,-83.114,176.441,23.088,153.651
C05299=1087.106,284.784,-83.087,176.439,23.085,153.651
C05300=1087.101,284.566,-83.062,176.437,23.083,153.651
C05301=1087.096,284.348,-83.036,176.434,23.079,153.651
C05302=1087.091,284.129,-83.010,176.432,23.077,153.650
C05303=1087.086,283.911,-82.984,176.429,23.073,153.650
C05304=1087.081,283.692,-82.958,176.427,23.071,153.650
C05305=1087.076,283.474,-82.931,176.423,23.068,153.650
C05306=1087.071,283.256,-82.905,176.421,23.065,153.649
C05307=1087.065,283.008,-82.876,176.418,23.062,153.649
C05308=1087.059,282.759,-82.847,176.415,23.059,153.649
C05309=1087.054,282.511,-82.817,176.412,23.056,153.648
C05310=1087.048,282.263,-82.788,176.410,23.052,153.648
C05311=1087.043,282.015,-82.759,176.407,23.049,153.648
C05312=1087.037,281.766,-82.729,176.404,23.046,153.647
C05313=1087.031,281.518,-82.700,176.401,23.043,153.647
C05314=1087.025,281.270,-82.670,176.398,23.040,153.647
C05315=1087.020,281.022,-82.641,176.395,23.036,153.647
C05316=1087.014,280.774,-82.612,176.392,23.033,153.646
C05317=1087.009,280.526,-82.582,176.390,23.030,153.646
C05318=1087.002,280.277,-82.553,176.387,23.027,153.646
C05319=1086.997,280.029,-82.524,176.384,23.024,153.645
C05320=1086.991,279.780,-82.495,176.381,23.021,153.645
C05321=1086.986,279.532,-82.466,176.378,23.017,153.645
C05322=1086.980,279.284,-82.437,176.375,23.014,153.644
C05323=1086.974,279.036,-82.407,176.372,23.011,153.644
C05324=1086.968,278.788,-82.378,176.370,23.008,153.644
C05325=1086.963,278.540,-82.349,176.367,23.005,153.644
C05326=1086.957,278.291,-82.321,176.364,23.002,153.643
C05327=1086.952,278.043,-82.291,176.361,22.998,153.643
C05328=1086.945,277.795,-82.262,176.358,22.995,153.643
C05329=1086.941,277.547,-82.233,176.355,22.992,153.642
C05330=1086.934,277.299,-82.204,176.353,22.989,153.642
C05331=1086.929,277.080,-82.179,176.349,22.987,153.642
C05332=1086.924,276.861,-82.153,176.347,22.984,153.642
C05333=1086.919,276.644,-82.128,176.345,22.981,153.641
C05334=1086.915,276.425,-82.102,176.342,22.978,153.641
C05335=1086.909,276.206,-82.077,176.340,22.976,153.641
C05336=1086.904,275.988,-82.051,176.337,22.972,153.641
C05337=1086.900,275.770,-82.026,176.334,22.970,153.640
C05338=1086.894,275.552,-82.000,176.332,22.967,153.640
C05339=1086.888,275.303,-81.972,176.329,22.964,153.640
C05340=1086.883,275.056,-81.943,176.326,22.961,153.640
C05341=1086.877,274.807,-81.914,176.323,22.958,153.639
C05342=1086.872,274.558,-81.885,176.320,22.955,153.639
C05343=1086.866,274.311,-81.856,176.318,22.952,153.639
C05344=1086.860,274.062,-81.828,176.315,22.949,153.638
C05345=1086.855,273.814,-81.798,176.312,22.945,153.638
C05346=1086.849,273.566,-81.770,176.309,22.942,153.638
C05347=1086.843,273.318,-81.741,176.306,22.939,153.638
C05348=1086.837,273.069,-81.713,176.304,22.937,153.637
C05349=1086.832,272.821,-81.683,176.301,22.934,153.637
C05350=1086.826,272.572,-81.655,176.298,22.930,153.637
C05351=1086.820,272.324,-81.626,176.295,22.927,153.637
C05352=1086.815,272.076,-81.598,176.292,22.924,153.636
C05353=1086.809,271.828,-81.568,176.290,22.921,153.636
C05354=1086.804,271.580,-81.540,176.287,22.918,153.636
C05355=1086.798,271.331,-81.512,176.284,22.915,153.635
C05356=1086.792,271.083,-81.483,176.281,22.912,153.635
C05357=1086.786,270.835,-81.455,176.278,22.909,153.635
C05358=1086.780,270.587,-81.426,176.275,22.906,153.635
C05359=1086.775,270.338,-81.397,176.272,22.903,153.634
C05360=1086.770,270.089,-81.369,176.269,22.900,153.634
C05361=1086.763,269.841,-81.340,176.266,22.896,153.634
C05362=1086.758,269.593,-81.312,176.264,22.894,153.634
C05363=1086.752,269.345,-81.284,176.261,22.890,153.633
C05364=1086.746,269.097,-81.255,176.258,22.887,153.633
C05365=1086.740,268.848,-81.227,176.255,22.885,153.633
C05366=1086.735,268.600,-81.199,176.253,22.882,153.633
C05367=1086.730,268.351,-81.170,176.250,22.879,153.632
C05368=1086.724,268.103,-81.141,176.247,22.875,153.632
C05369=1086.718,267.855,-81.113,176.244,22.872,153.632
C05370=1086.712,267.606,-81.085,176.241,22.869,153.631
C05371=1086.707,267.358,-81.057,176.238,22.867,153.631
C05372=1086.701,267.110,-81.028,176.235,22.863,153.631
C05373=1086.696,266.861,-81.000,176.232,22.860,153.631
C05374=1086.690,266.613,-80.971,176.229,22.857,153.630
C05375=1086.684,266.365,-80.943,176.227,22.854,153.630
C05376=1086.678,266.117,-80.915,176.224,22.851,153.630
C05377=1086.673,265.868,-80.887,176.221,22.848,153.630
C05378=1086.667,265.620,-80.859,176.218,22.845,153.629
C05379=1086.662,265.372,-80.831,176.216,22.842,153.629
C05380=1086.656,265.123,-80.802,176.213,22.839,153.629
C05381=1086.650,264.875,-80.775,176.210,22.836,153.629
C05382=1086.644,264.626,-80.746,176.207,22.833,153.628
C05383=1086.639,264.378,-80.718,176.205,22.830,153.628
C05384=1086.633,264.129,-80.690,176.202,22.827,153.628
C05385=1086.628,263.881,-80.662,176.199,22.824,153.628
C05386=1086.621,263.633,-80.634,176.196,22.822,153.627
C05387=1086.613,263.259,-80.592,176.192,22.817,153.627
C05388=1086.604,262.884,-80.550,176.187,22.813,153.627
C05389=1086.595,262.510,-80.507,176.183,22.808,153.626
C05390=1086.586,262.136,-80.466,176.179,22.804,153.626
C05391=1086.580,261.887,-80.438,176.176,22.801,153.626
C05392=1086.575,261.639,-80.410,176.174,22.798,153.625
C05393=1086.569,261.390,-80.381,176.170,22.795,153.625
C05394=1086.563,261.142,-80.355,176.167,22.792,153.625
C05395=1086.557,260.893,-80.326,176.164,22.789,153.625
C05396=1086.552,260.645,-80.298,176.162,22.786,153.625
C05397=1086.545,260.397,-80.271,176.159,22.783,153.624
C05398=1086.540,260.149,-80.243,176.156,22.780,153.624
C05399=1086.535,259.900,-80.215,176.154,22.778,153.624
C05400=1086.529,259.651,-80.187,176.151,22.774,153.624
C05401=1086.523,259.404,-80.160,176.148,22.771,153.623
C05402=1086.517,259.155,-80.131,176.145,22.768,153.623
C05403=1086.512,258.906,-80.104,176.142,22.766,153.623
C05404=1086.506,258.659,-80.077,176.139,22.762,153.623
C05405=1086.500,258.410,-80.048,176.136,22.760,153.622
C05406=1086.495,258.161,-80.021,176.134,22.757,153.622
C05407=1086.488,257.913,-79.993,176.131,22.754,153.622
C05408=1086.483,257.665,-79.965,176.128,22.751,153.622
C05409=1086.477,257.416,-79.939,176.126,22.748,153.621
C05410=1086.471,257.167,-79.911,176.123,22.745,153.621
C05411=1086.466,256.919,-79.883,176.120,22.742,153.621
C05412=1086.460,256.671,-79.856,176.117,22.739,153.621
C05413=1086.454,256.422,-79.828,176.115,22.736,153.620
C05414=1086.449,256.174,-79.800,176.112,22.733,153.620
C05415=1086.443,255.926,-79.773,176.108,22.730,153.620
C05416=1086.437,255.677,-79.745,176.106,22.728,153.620
C05417=1086.431,255.429,-79.718,176.103,22.724,153.619
C05418=1086.426,255.180,-79.691,176.100,22.722,153.619
C05419=1086.421,254.932,-79.663,176.098,22.719,153.619
C05420=1086.414,254.683,-79.636,176.095,22.716,153.619
C05421=1086.409,254.435,-79.608,176.092,22.713,153.619
C05422=1086.403,254.187,-79.581,176.090,22.710,153.618
C05423=1086.397,253.938,-79.553,176.087,22.707,153.618
C05424=1086.392,253.689,-79.526,176.084,22.704,153.618
C05425=1086.386,253.441,-79.498,176.081,22.701,153.617
C05426=1086.381,253.193,-79.471,176.078,22.698,153.617
C05427=1086.375,252.944,-79.444,176.075,22.695,153.617
C05428=1086.369,252.696,-79.416,176.073,22.693,153.617
C05429=1086.364,252.447,-79.389,176.070,22.689,153.617
C05430=1086.359,252.199,-79.362,176.067,22.686,153.616
C05431=1086.353,251.951,-79.335,176.065,22.684,153.616
C05432=1086.347,251.701,-79.307,176.062,22.681,153.616
C05433=1086.341,251.453,-79.281,176.059,22.677,153.616
C05434=1086.336,251.205,-79.253,176.057,22.675,153.615
C05435=1086.330,250.957,-79.226,176.054,22.672,153.615
C05436=1086.325,250.708,-79.199,176.051,22.669,153.615
C05437=1086.319,250.460,-79.171,176.048,22.666,153.614
C05438=1086.313,250.211,-79.144,176.045,22.663,153.614
C05439=1086.305,249.834,-79.103,176.042,22.659,153.614
C05440=1086.297,249.457,-79.061,176.037,22.654,153.614
C05441=1086.288,249.080,-79.021,176.033,22.649,153.613
C05442=1086.280,248.702,-78.980,176.029,22.645,153.613
C05443=1086.275,248.454,-78.953,176.026,22.642,153.613
C05444=1086.269,248.206,-78.925,176.024,22.639,153.612
C05445=1086.264,247.957,-78.898,176.021,22.636,153.612
C05446=1086.258,247.709,-78.871,176.018,22.633,153.612
C05447=1086.253,247.460,-78.844,176.016,22.630,153.612
